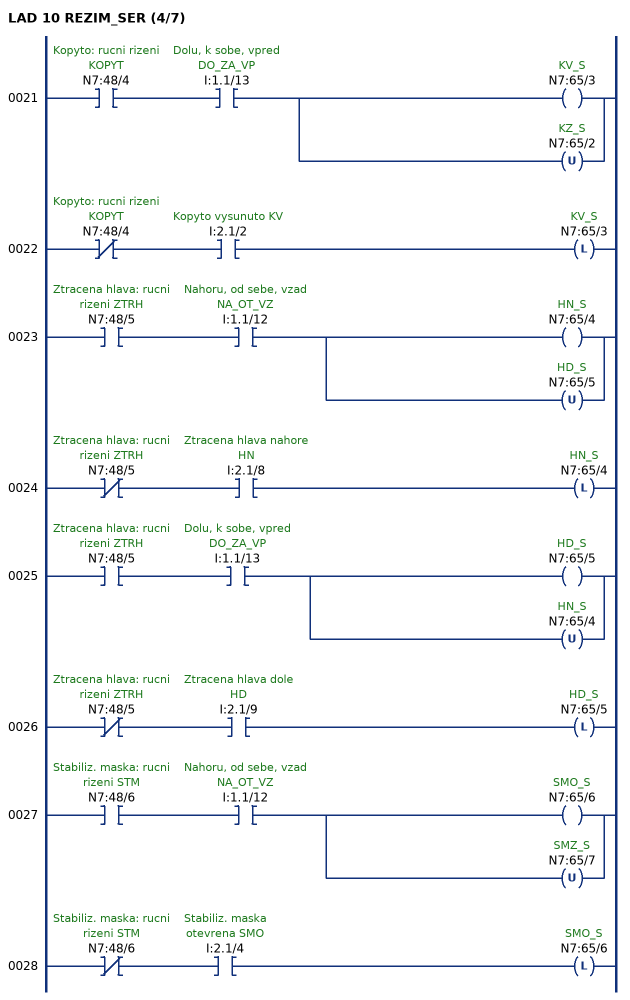
% Rung: 21 %
SOR XIC N7:48/4 XIC I:1.1/13 BST OTE N7:65/3 NXB OTU N7:65/2 BND EOR
%   N7:48/4  KOPYT  "Kopyto: rucni rizeni" %
%   I:1.1/13  DO_ZA_VP  "Dolu, k sobe, vpred" %
%   N7:65/3  KV_S %
%   N7:65/2  KZ_S %
% Rung: 22 %
SOR XIO N7:48/4 XIC I:2.1/2 OTL N7:65/3 EOR
%   N7:48/4  KOPYT  "Kopyto: rucni rizeni" %
%   I:2.1/2  KV  "Kopyto vysunuto" %
%   N7:65/3  KV_S %
% Rung: 23 %
SOR XIC N7:48/5 XIC I:1.1/12 BST OTE N7:65/4 NXB OTU N7:65/5 BND EOR
%   N7:48/5  ZTRH  "Ztracena hlava: rucni rizeni" %
%   I:1.1/12  NA_OT_VZ  "Nahoru, od sebe, vzad" %
%   N7:65/4  HN_S %
%   N7:65/5  HD_S %
% Rung: 24 %
SOR XIO N7:48/5 XIC I:2.1/8 OTL N7:65/4 EOR
%   N7:48/5  ZTRH  "Ztracena hlava: rucni rizeni" %
%   I:2.1/8  HN  "Ztracena hlava nahore" %
%   N7:65/4  HN_S %
% Rung: 25 %
SOR XIC N7:48/5 XIC I:1.1/13 BST OTE N7:65/5 NXB OTU N7:65/4 BND EOR
%   N7:48/5  ZTRH  "Ztracena hlava: rucni rizeni" %
%   I:1.1/13  DO_ZA_VP  "Dolu, k sobe, vpred" %
%   N7:65/5  HD_S %
%   N7:65/4  HN_S %
% Rung: 26 %
SOR XIO N7:48/5 XIC I:2.1/9 OTL N7:65/5 EOR
%   N7:48/5  ZTRH  "Ztracena hlava: rucni rizeni" %
%   I:2.1/9  HD  "Ztracena hlava dole" %
%   N7:65/5  HD_S %
% Rung: 27 %
SOR XIC N7:48/6 XIC I:1.1/12 BST OTE N7:65/6 NXB OTU N7:65/7 BND EOR
%   N7:48/6  STM  "Stabiliz. maska: rucni rizeni" %
%   I:1.1/12  NA_OT_VZ  "Nahoru, od sebe, vzad" %
%   N7:65/6  SMO_S %
%   N7:65/7  SMZ_S %
% Rung: 28 %
SOR XIO N7:48/6 XIC I:2.1/4 OTL N7:65/6 EOR
%   N7:48/6  STM  "Stabiliz. maska: rucni rizeni" %
%   I:2.1/4  SMO  "Stabiliz. maska otevrena" %
%   N7:65/6  SMO_S %

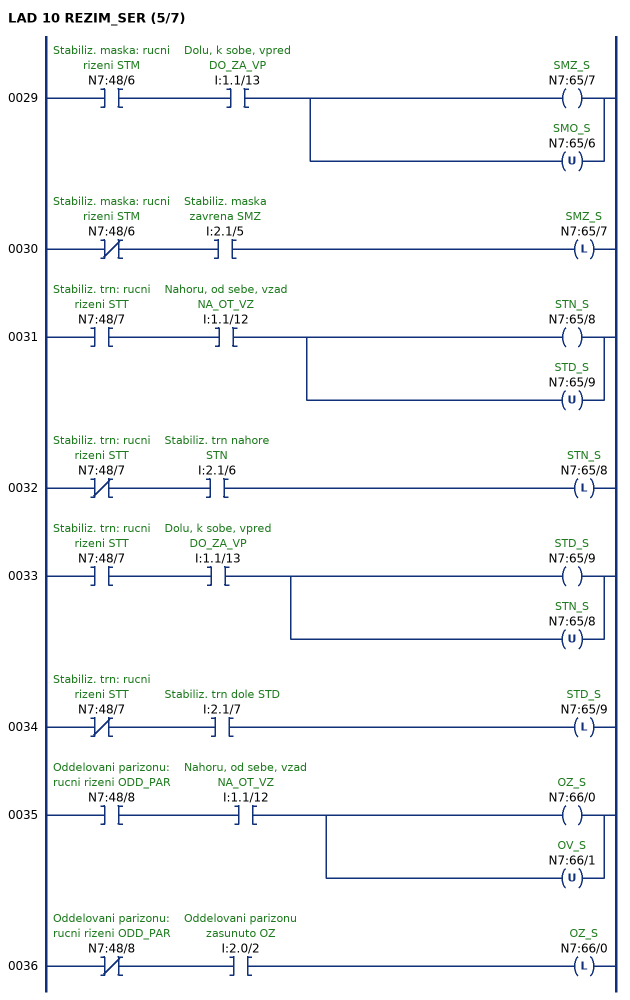
% Rung: 29 %
SOR XIC N7:48/6 XIC I:1.1/13 BST OTE N7:65/7 NXB OTU N7:65/6 BND EOR
%   N7:48/6  STM  "Stabiliz. maska: rucni rizeni" %
%   I:1.1/13  DO_ZA_VP  "Dolu, k sobe, vpred" %
%   N7:65/7  SMZ_S %
%   N7:65/6  SMO_S %
% Rung: 30 %
SOR XIO N7:48/6 XIC I:2.1/5 OTL N7:65/7 EOR
%   N7:48/6  STM  "Stabiliz. maska: rucni rizeni" %
%   I:2.1/5  SMZ  "Stabiliz. maska zavrena" %
%   N7:65/7  SMZ_S %
% Rung: 31 %
SOR XIC N7:48/7 XIC I:1.1/12 BST OTE N7:65/8 NXB OTU N7:65/9 BND EOR
%   N7:48/7  STT  "Stabiliz. trn: rucni rizeni" %
%   I:1.1/12  NA_OT_VZ  "Nahoru, od sebe, vzad" %
%   N7:65/8  STN_S %
%   N7:65/9  STD_S %
% Rung: 32 %
SOR XIO N7:48/7 XIC I:2.1/6 OTL N7:65/8 EOR
%   N7:48/7  STT  "Stabiliz. trn: rucni rizeni" %
%   I:2.1/6  STN  "Stabiliz. trn nahore" %
%   N7:65/8  STN_S %
% Rung: 33 %
SOR XIC N7:48/7 XIC I:1.1/13 BST OTE N7:65/9 NXB OTU N7:65/8 BND EOR
%   N7:48/7  STT  "Stabiliz. trn: rucni rizeni" %
%   I:1.1/13  DO_ZA_VP  "Dolu, k sobe, vpred" %
%   N7:65/9  STD_S %
%   N7:65/8  STN_S %
% Rung: 34 %
SOR XIO N7:48/7 XIC I:2.1/7 OTL N7:65/9 EOR
%   N7:48/7  STT  "Stabiliz. trn: rucni rizeni" %
%   I:2.1/7  STD  "Stabiliz. trn dole" %
%   N7:65/9  STD_S %
% Rung: 35 %
SOR XIC N7:48/8 XIC I:1.1/12 BST OTE N7:66/0 NXB OTU N7:66/1 BND EOR
%   N7:48/8  ODD_PAR  "Oddelovani parizonu: rucni rizeni" %
%   I:1.1/12  NA_OT_VZ  "Nahoru, od sebe, vzad" %
%   N7:66/0  OZ_S %
%   N7:66/1  OV_S %
% Rung: 36 %
SOR XIO N7:48/8 XIC I:2.0/2 OTL N7:66/0 EOR
%   N7:48/8  ODD_PAR  "Oddelovani parizonu: rucni rizeni" %
%   I:2.0/2  OZ  "Oddelovani parizonu zasunuto" %
%   N7:66/0  OZ_S %

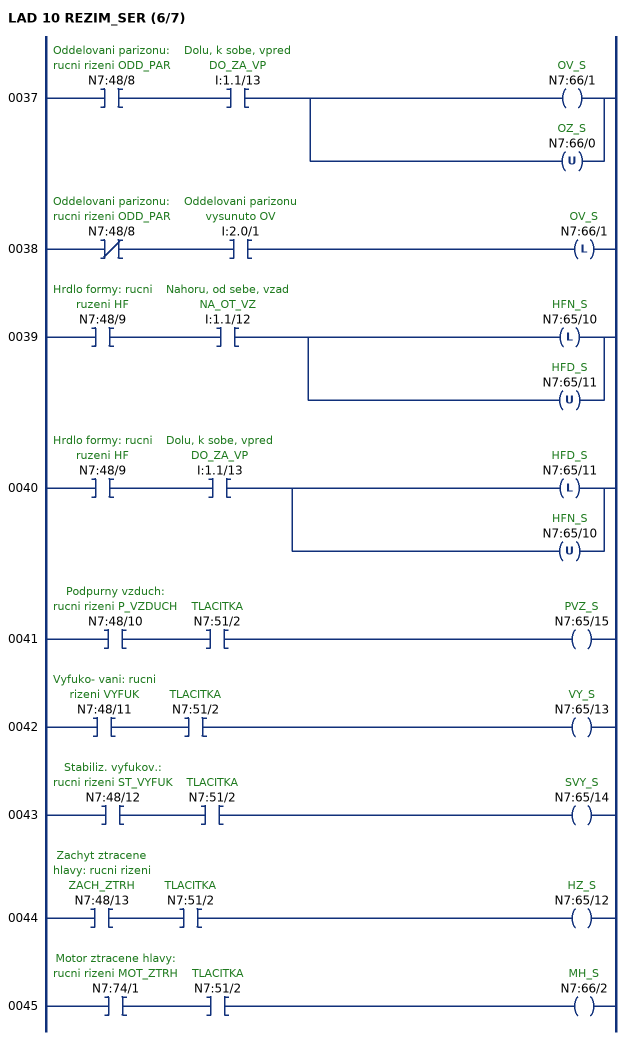
% Rung: 37 %
SOR XIC N7:48/8 XIC I:1.1/13 BST OTE N7:66/1 NXB OTU N7:66/0 BND EOR
%   N7:48/8  ODD_PAR  "Oddelovani parizonu: rucni rizeni" %
%   I:1.1/13  DO_ZA_VP  "Dolu, k sobe, vpred" %
%   N7:66/1  OV_S %
%   N7:66/0  OZ_S %
% Rung: 38 %
SOR XIO N7:48/8 XIC I:2.0/1 OTL N7:66/1 EOR
%   N7:48/8  ODD_PAR  "Oddelovani parizonu: rucni rizeni" %
%   I:2.0/1  OV  "Oddelovani parizonu vysunuto" %
%   N7:66/1  OV_S %
% Rung: 39 %
SOR XIC N7:48/9 XIC I:1.1/12 BST OTL N7:65/10 NXB OTU N7:65/11 BND EOR
%   N7:48/9  HF  "Hrdlo formy: rucni ruzeni" %
%   I:1.1/12  NA_OT_VZ  "Nahoru, od sebe, vzad" %
%   N7:65/10  HFN_S %
%   N7:65/11  HFD_S %
% Rung: 40 %
SOR XIC N7:48/9 XIC I:1.1/13 BST OTL N7:65/11 NXB OTU N7:65/10 BND EOR
%   N7:48/9  HF  "Hrdlo formy: rucni ruzeni" %
%   I:1.1/13  DO_ZA_VP  "Dolu, k sobe, vpred" %
%   N7:65/11  HFD_S %
%   N7:65/10  HFN_S %
% Rung: 41 %
SOR XIC N7:48/10 XIC N7:51/2 OTE N7:65/15 EOR
%   N7:48/10  P_VZDUCH  "Podpurny vzduch: rucni rizeni" %
%   N7:51/2  TLACITKA %
%   N7:65/15  PVZ_S %
% Rung: 42 %
SOR XIC N7:48/11 XIC N7:51/2 OTE N7:65/13 EOR
%   N7:48/11  VYFUK  "Vyfuko- vani: rucni rizeni" %
%   N7:51/2  TLACITKA %
%   N7:65/13  VY_S %
% Rung: 43 %
SOR XIC N7:48/12 XIC N7:51/2 OTE N7:65/14 EOR
%   N7:48/12  ST_VYFUK  "Stabiliz. vyfukov.: rucni rizeni" %
%   N7:51/2  TLACITKA %
%   N7:65/14  SVY_S %
% Rung: 44 %
SOR XIC N7:48/13 XIC N7:51/2 OTE N7:65/12 EOR
%   N7:48/13  ZACH_ZTRH  "Zachyt ztracene hlavy: rucni rizeni" %
%   N7:51/2  TLACITKA %
%   N7:65/12  HZ_S %
% Rung: 45 %
SOR XIC N7:74/1 XIC N7:51/2 OTE N7:66/2 EOR
%   N7:74/1  MOT_ZTRH  "Motor ztracene hlavy: rucni rizeni" %
%   N7:51/2  TLACITKA %
%   N7:66/2  MH_S %

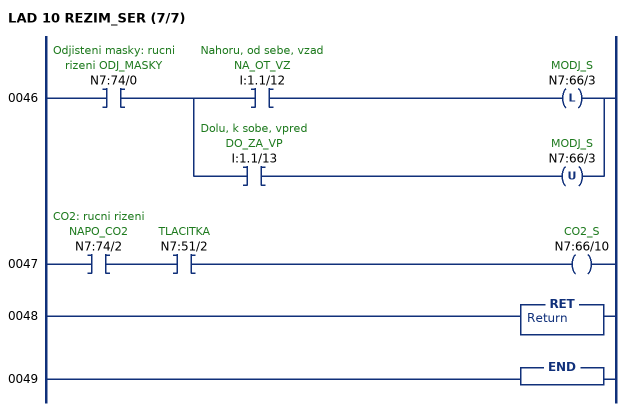
% Rung: 46 %
SOR XIC N7:74/0 BST XIC I:1.1/12 OTL N7:66/3 NXB XIC I:1.1/13 OTU N7:66/3 BND EOR
%   N7:74/0  ODJ_MASKY  "Odjisteni masky: rucni rizeni" %
%   I:1.1/12  NA_OT_VZ  "Nahoru, od sebe, vzad" %
%   N7:66/3  MODJ_S %
%   I:1.1/13  DO_ZA_VP  "Dolu, k sobe, vpred" %
% Rung: 47 %
SOR XIC N7:74/2 XIC N7:51/2 OTE N7:66/10 EOR
%   N7:74/2  NAPO_CO2  "CO2: rucni rizeni" %
%   N7:51/2  TLACITKA %
%   N7:66/10  CO2_S %
% Rung: 48 %
SOR RET EOR
% Rung: 49 %
SOR END EOR

LADDER 11 "REZIM_RUC"
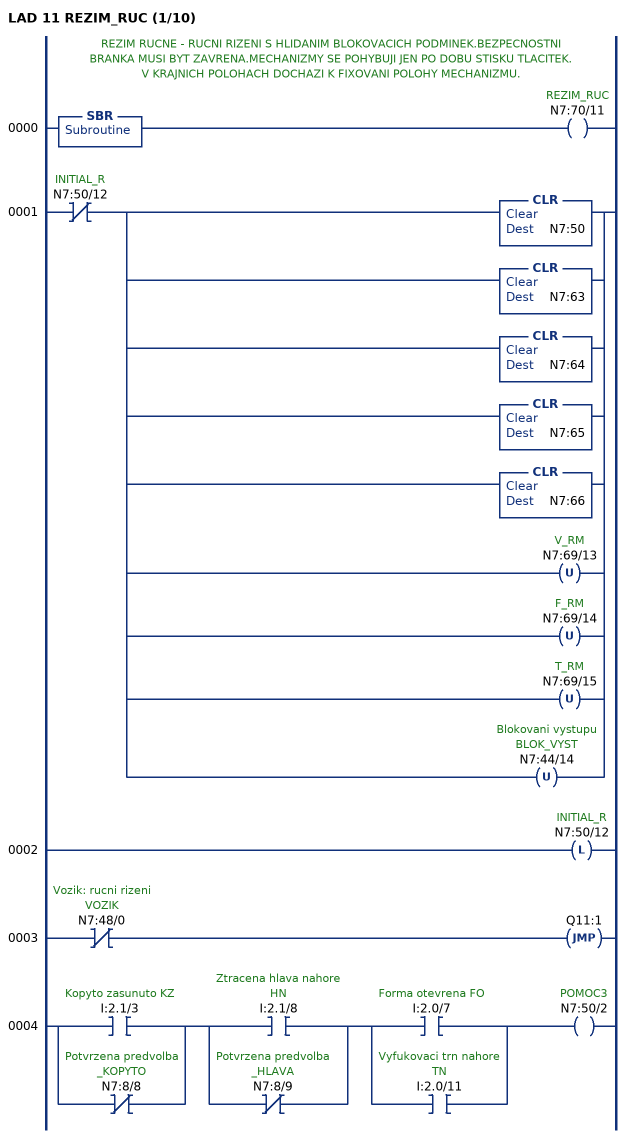
% Rung: 0 %
% REZIM RUCNE - RUCNI RIZENI S HLIDANIM BLOKOVACICH PODMINEK.BEZPECNOSTNI
% BRANKA MUSI BYT ZAVRENA.MECHANIZMY SE POHYBUJI JEN PO DOBU STISKU TLACITEK.
% V KRAJNICH POLOHACH DOCHAZI K FIXOVANI POLOHY MECHANIZMU. %
SOR SBR OTE N7:70/11 EOR
%   N7:70/11  REZIM_RUC %
% Rung: 1 %
SOR XIO N7:50/12 BST CLR N7:50 NXB CLR N7:63 NXB CLR N7:64 NXB CLR N7:65 NXB CLR N7:66 NXB OTU N7:69/13 NXB OTU N7:69/14 NXB OTU N7:69/15 NXB OTU N7:44/14 BND EOR
%   N7:50/12  INITIAL_R %
%   CLR N7:50  "Pomocne merkry" %
%   CLR N7:63  "Merkry vystupu rucniho rezimu" %
%   CLR N7:64  "Merkry vystupu rucniho rezimu" %
%   CLR N7:65  "Merkry vystupu rezimu serizovani" %
%   CLR N7:66  "Merkry vystupu rezimu serizovani" %
%   N7:69/13  V_RM %
%   N7:69/14  F_RM %
%   N7:69/15  T_RM %
%   N7:44/14  BLOK_VYST  "Blokovani vystupu" %
% Rung: 2 %
SOR OTL N7:50/12 EOR
%   N7:50/12  INITIAL_R %
% Rung: 3 %
SOR XIO N7:48/0 JMP Q11:1 EOR
%   N7:48/0  VOZIK  "Vozik: rucni rizeni" %
% Rung: 4 %
SOR BST XIC I:2.1/3 NXB XIO N7:8/8 BND BST XIC I:2.1/8 NXB XIO N7:8/9 BND BST XIC I:2.0/7 NXB XIC I:2.0/11 BND OTE N7:50/2 EOR
%   I:2.1/3  KZ  "Kopyto zasunuto" %
%   N7:8/8  _KOPYTO  "Potvrzena predvolba" %
%   I:2.1/8  HN  "Ztracena hlava nahore" %
%   N7:8/9  _HLAVA  "Potvrzena predvolba" %
%   I:2.0/7  FO  "Forma otevrena" %
%   I:2.0/11  TN  "Vyfukovaci trn nahore" %
%   N7:50/2  POMOC3 %

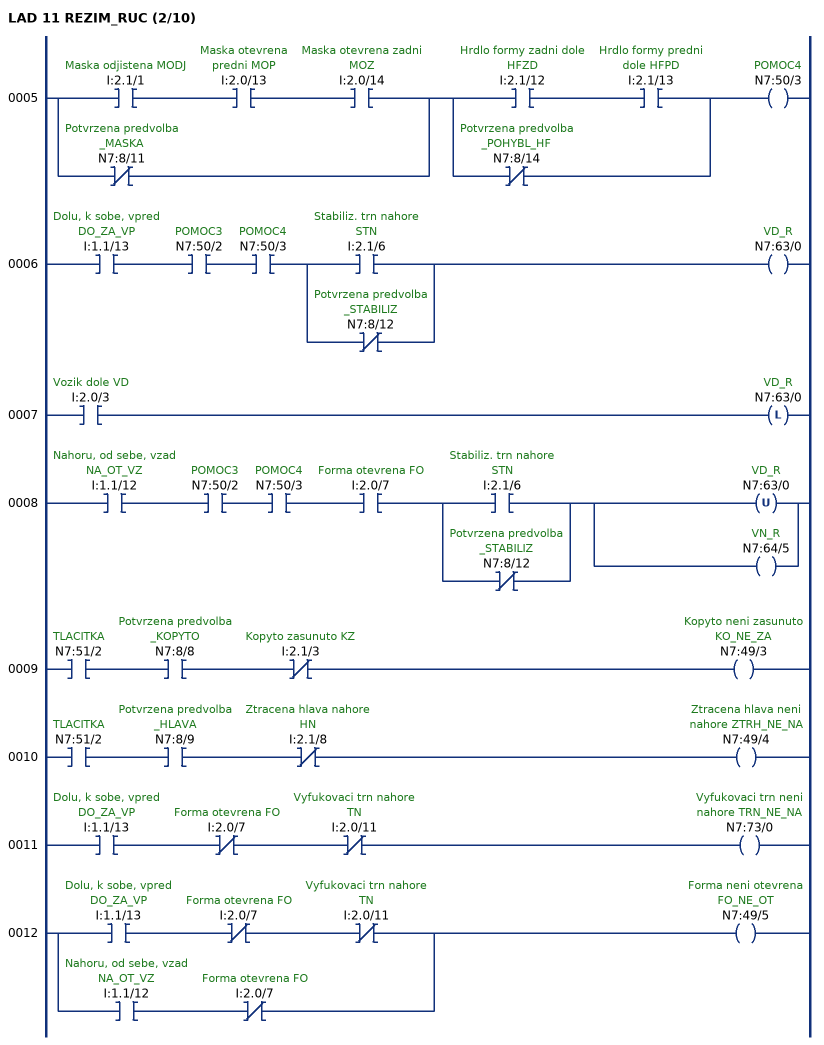
% Rung: 5 %
SOR BST XIC I:2.1/1 XIC I:2.0/13 XIC I:2.0/14 NXB XIO N7:8/11 BND BST XIC I:2.1/12 XIC I:2.1/13 NXB XIO N7:8/14 BND OTE N7:50/3 EOR
%   I:2.1/1  MODJ  "Maska odjistena" %
%   I:2.0/13  MOP  "Maska otevrena predni" %
%   I:2.0/14  MOZ  "Maska otevrena zadni" %
%   N7:8/11  _MASKA  "Potvrzena predvolba" %
%   I:2.1/12  HFZD  "Hrdlo formy zadni dole" %
%   I:2.1/13  HFPD  "Hrdlo formy predni dole" %
%   N7:8/14  _POHYBL_HF  "Potvrzena predvolba" %
%   N7:50/3  POMOC4 %
% Rung: 6 %
SOR XIC I:1.1/13 XIC N7:50/2 XIC N7:50/3 BST XIC I:2.1/6 NXB XIO N7:8/12 BND OTE N7:63/0 EOR
%   I:1.1/13  DO_ZA_VP  "Dolu, k sobe, vpred" %
%   N7:50/2  POMOC3 %
%   N7:50/3  POMOC4 %
%   I:2.1/6  STN  "Stabiliz. trn nahore" %
%   N7:8/12  _STABILIZ  "Potvrzena predvolba" %
%   N7:63/0  VD_R %
% Rung: 7 %
SOR XIC I:2.0/3 OTL N7:63/0 EOR
%   I:2.0/3  VD  "Vozik dole" %
%   N7:63/0  VD_R %
% Rung: 8 %
SOR XIC I:1.1/12 XIC N7:50/2 XIC N7:50/3 XIC I:2.0/7 BST XIC I:2.1/6 NXB XIO N7:8/12 BND BST OTU N7:63/0 NXB OTE N7:64/5 BND EOR
%   I:1.1/12  NA_OT_VZ  "Nahoru, od sebe, vzad" %
%   N7:50/2  POMOC3 %
%   N7:50/3  POMOC4 %
%   I:2.0/7  FO  "Forma otevrena" %
%   I:2.1/6  STN  "Stabiliz. trn nahore" %
%   N7:8/12  _STABILIZ  "Potvrzena predvolba" %
%   N7:63/0  VD_R %
%   N7:64/5  VN_R %
% Rung: 9 %
SOR XIC N7:51/2 XIC N7:8/8 XIO I:2.1/3 OTE N7:49/3 EOR
%   N7:51/2  TLACITKA %
%   N7:8/8  _KOPYTO  "Potvrzena predvolba" %
%   I:2.1/3  KZ  "Kopyto zasunuto" %
%   N7:49/3  KO_NE_ZA  "Kopyto neni zasunuto" %
% Rung: 10 %
SOR XIC N7:51/2 XIC N7:8/9 XIO I:2.1/8 OTE N7:49/4 EOR
%   N7:51/2  TLACITKA %
%   N7:8/9  _HLAVA  "Potvrzena predvolba" %
%   I:2.1/8  HN  "Ztracena hlava nahore" %
%   N7:49/4  ZTRH_NE_NA  "Ztracena hlava neni nahore" %
% Rung: 11 %
SOR XIC I:1.1/13 XIO I:2.0/7 XIO I:2.0/11 OTE N7:73/0 EOR
%   I:1.1/13  DO_ZA_VP  "Dolu, k sobe, vpred" %
%   I:2.0/7  FO  "Forma otevrena" %
%   I:2.0/11  TN  "Vyfukovaci trn nahore" %
%   N7:73/0  TRN_NE_NA  "Vyfukovaci trn neni nahore" %
% Rung: 12 %
SOR BST XIC I:1.1/13 XIO I:2.0/7 XIO I:2.0/11 NXB XIC I:1.1/12 XIO I:2.0/7 BND OTE N7:49/5 EOR
%   I:1.1/13  DO_ZA_VP  "Dolu, k sobe, vpred" %
%   I:2.0/7  FO  "Forma otevrena" %
%   I:2.0/11  TN  "Vyfukovaci trn nahore" %
%   I:1.1/12  NA_OT_VZ  "Nahoru, od sebe, vzad" %
%   N7:49/5  FO_NE_OT  "Forma neni otevrena" %

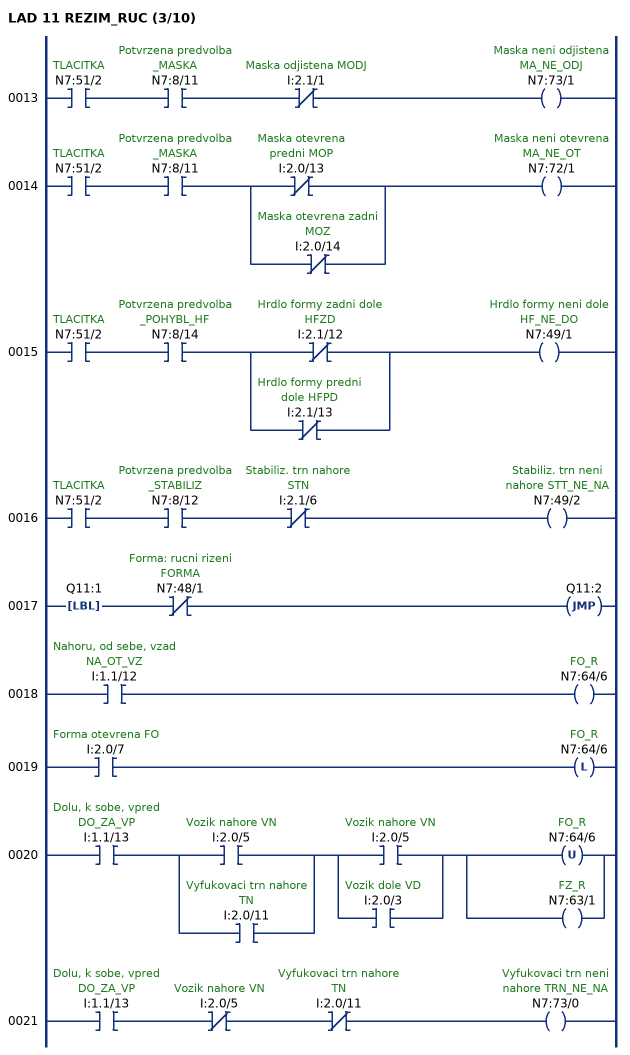
% Rung: 13 %
SOR XIC N7:51/2 XIC N7:8/11 XIO I:2.1/1 OTE N7:73/1 EOR
%   N7:51/2  TLACITKA %
%   N7:8/11  _MASKA  "Potvrzena predvolba" %
%   I:2.1/1  MODJ  "Maska odjistena" %
%   N7:73/1  MA_NE_ODJ  "Maska neni odjistena" %
% Rung: 14 %
SOR XIC N7:51/2 XIC N7:8/11 BST XIO I:2.0/13 NXB XIO I:2.0/14 BND OTE N7:72/1 EOR
%   N7:51/2  TLACITKA %
%   N7:8/11  _MASKA  "Potvrzena predvolba" %
%   I:2.0/13  MOP  "Maska otevrena predni" %
%   I:2.0/14  MOZ  "Maska otevrena zadni" %
%   N7:72/1  MA_NE_OT  "Maska neni otevrena" %
% Rung: 15 %
SOR XIC N7:51/2 XIC N7:8/14 BST XIO I:2.1/12 NXB XIO I:2.1/13 BND OTE N7:49/1 EOR
%   N7:51/2  TLACITKA %
%   N7:8/14  _POHYBL_HF  "Potvrzena predvolba" %
%   I:2.1/12  HFZD  "Hrdlo formy zadni dole" %
%   I:2.1/13  HFPD  "Hrdlo formy predni dole" %
%   N7:49/1  HF_NE_DO  "Hrdlo formy neni dole" %
% Rung: 16 %
SOR XIC N7:51/2 XIC N7:8/12 XIO I:2.1/6 OTE N7:49/2 EOR
%   N7:51/2  TLACITKA %
%   N7:8/12  _STABILIZ  "Potvrzena predvolba" %
%   I:2.1/6  STN  "Stabiliz. trn nahore" %
%   N7:49/2  STT_NE_NA  "Stabiliz. trn neni nahore" %
% Rung: 17 %
SOR LBL Q11:1 XIO N7:48/1 JMP Q11:2 EOR
%   N7:48/1  FORMA  "Forma: rucni rizeni" %
% Rung: 18 %
SOR XIC I:1.1/12 OTE N7:64/6 EOR
%   I:1.1/12  NA_OT_VZ  "Nahoru, od sebe, vzad" %
%   N7:64/6  FO_R %
% Rung: 19 %
SOR XIC I:2.0/7 OTL N7:64/6 EOR
%   I:2.0/7  FO  "Forma otevrena" %
%   N7:64/6  FO_R %
% Rung: 20 %
SOR XIC I:1.1/13 BST XIC I:2.0/5 NXB XIC I:2.0/11 BND BST XIC I:2.0/5 NXB XIC I:2.0/3 BND BST OTU N7:64/6 NXB OTE N7:63/1 BND EOR
%   I:1.1/13  DO_ZA_VP  "Dolu, k sobe, vpred" %
%   I:2.0/5  VN  "Vozik nahore" %
%   I:2.0/11  TN  "Vyfukovaci trn nahore" %
%   I:2.0/3  VD  "Vozik dole" %
%   N7:64/6  FO_R %
%   N7:63/1  FZ_R %
% Rung: 21 %
SOR XIC I:1.1/13 XIO I:2.0/5 XIO I:2.0/11 OTE N7:73/0 EOR
%   I:1.1/13  DO_ZA_VP  "Dolu, k sobe, vpred" %
%   I:2.0/5  VN  "Vozik nahore" %
%   I:2.0/11  TN  "Vyfukovaci trn nahore" %
%   N7:73/0  TRN_NE_NA  "Vyfukovaci trn neni nahore" %

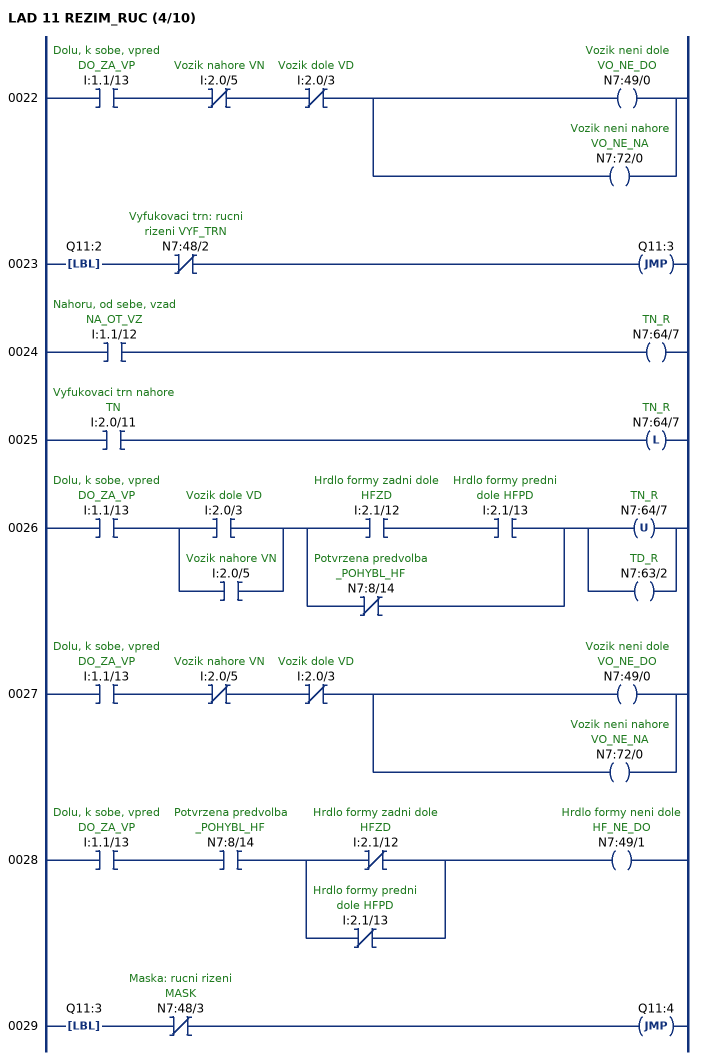
% Rung: 22 %
SOR XIC I:1.1/13 XIO I:2.0/5 XIO I:2.0/3 BST OTE N7:49/0 NXB OTE N7:72/0 BND EOR
%   I:1.1/13  DO_ZA_VP  "Dolu, k sobe, vpred" %
%   I:2.0/5  VN  "Vozik nahore" %
%   I:2.0/3  VD  "Vozik dole" %
%   N7:49/0  VO_NE_DO  "Vozik neni dole" %
%   N7:72/0  VO_NE_NA  "Vozik neni nahore" %
% Rung: 23 %
SOR LBL Q11:2 XIO N7:48/2 JMP Q11:3 EOR
%   N7:48/2  VYF_TRN  "Vyfukovaci trn: rucni rizeni" %
% Rung: 24 %
SOR XIC I:1.1/12 OTE N7:64/7 EOR
%   I:1.1/12  NA_OT_VZ  "Nahoru, od sebe, vzad" %
%   N7:64/7  TN_R %
% Rung: 25 %
SOR XIC I:2.0/11 OTL N7:64/7 EOR
%   I:2.0/11  TN  "Vyfukovaci trn nahore" %
%   N7:64/7  TN_R %
% Rung: 26 %
SOR XIC I:1.1/13 BST XIC I:2.0/3 NXB XIC I:2.0/5 BND BST XIC I:2.1/12 XIC I:2.1/13 NXB XIO N7:8/14 BND BST OTU N7:64/7 NXB OTE N7:63/2 BND EOR
%   I:1.1/13  DO_ZA_VP  "Dolu, k sobe, vpred" %
%   I:2.0/3  VD  "Vozik dole" %
%   I:2.0/5  VN  "Vozik nahore" %
%   I:2.1/12  HFZD  "Hrdlo formy zadni dole" %
%   I:2.1/13  HFPD  "Hrdlo formy predni dole" %
%   N7:8/14  _POHYBL_HF  "Potvrzena predvolba" %
%   N7:64/7  TN_R %
%   N7:63/2  TD_R %
% Rung: 27 %
SOR XIC I:1.1/13 XIO I:2.0/5 XIO I:2.0/3 BST OTE N7:49/0 NXB OTE N7:72/0 BND EOR
%   I:1.1/13  DO_ZA_VP  "Dolu, k sobe, vpred" %
%   I:2.0/5  VN  "Vozik nahore" %
%   I:2.0/3  VD  "Vozik dole" %
%   N7:49/0  VO_NE_DO  "Vozik neni dole" %
%   N7:72/0  VO_NE_NA  "Vozik neni nahore" %
% Rung: 28 %
SOR XIC I:1.1/13 XIC N7:8/14 BST XIO I:2.1/12 NXB XIO I:2.1/13 BND OTE N7:49/1 EOR
%   I:1.1/13  DO_ZA_VP  "Dolu, k sobe, vpred" %
%   N7:8/14  _POHYBL_HF  "Potvrzena predvolba" %
%   I:2.1/12  HFZD  "Hrdlo formy zadni dole" %
%   I:2.1/13  HFPD  "Hrdlo formy predni dole" %
%   N7:49/1  HF_NE_DO  "Hrdlo formy neni dole" %
% Rung: 29 %
SOR LBL Q11:3 XIO N7:48/3 JMP Q11:4 EOR
%   N7:48/3  MASK  "Maska: rucni rizeni" %

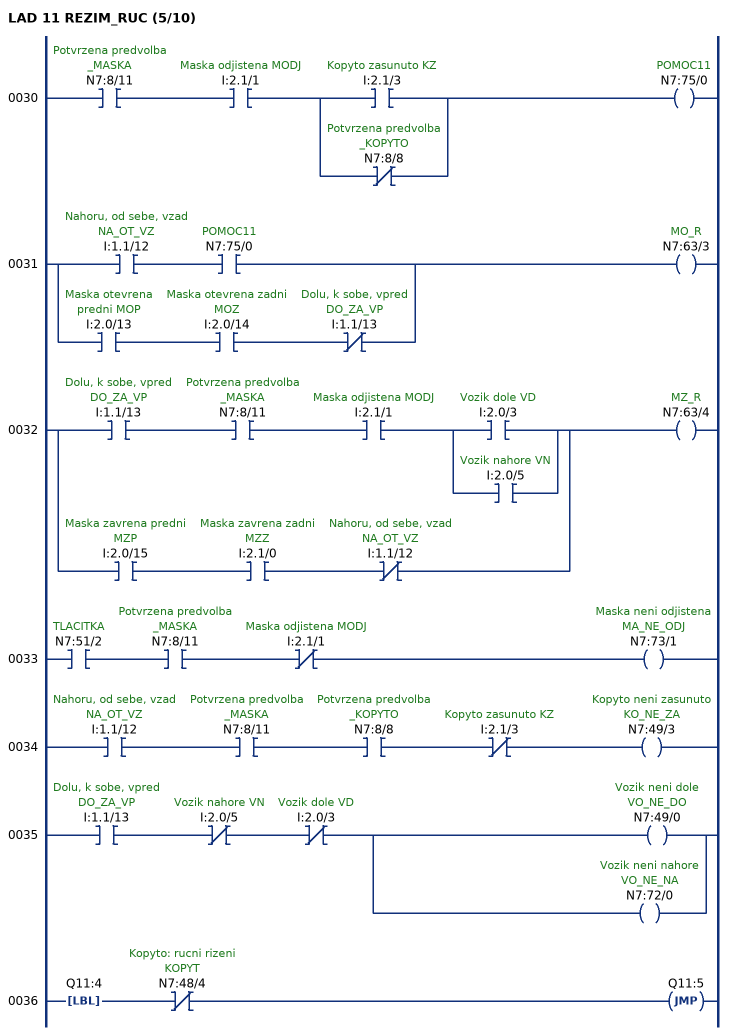
% Rung: 30 %
SOR XIC N7:8/11 XIC I:2.1/1 BST XIC I:2.1/3 NXB XIO N7:8/8 BND OTE N7:75/0 EOR
%   N7:8/11  _MASKA  "Potvrzena predvolba" %
%   I:2.1/1  MODJ  "Maska odjistena" %
%   I:2.1/3  KZ  "Kopyto zasunuto" %
%   N7:8/8  _KOPYTO  "Potvrzena predvolba" %
%   N7:75/0  POMOC11 %
% Rung: 31 %
SOR BST XIC I:1.1/12 XIC N7:75/0 NXB XIC I:2.0/13 XIC I:2.0/14 XIO I:1.1/13 BND OTE N7:63/3 EOR
%   I:1.1/12  NA_OT_VZ  "Nahoru, od sebe, vzad" %
%   N7:75/0  POMOC11 %
%   I:2.0/13  MOP  "Maska otevrena predni" %
%   I:2.0/14  MOZ  "Maska otevrena zadni" %
%   I:1.1/13  DO_ZA_VP  "Dolu, k sobe, vpred" %
%   N7:63/3  MO_R %
% Rung: 32 %
SOR BST XIC I:1.1/13 XIC N7:8/11 XIC I:2.1/1 BST XIC I:2.0/3 NXB XIC I:2.0/5 BND NXB XIC I:2.0/15 XIC I:2.1/0 XIO I:1.1/12 BND OTE N7:63/4 EOR
%   I:1.1/13  DO_ZA_VP  "Dolu, k sobe, vpred" %
%   N7:8/11  _MASKA  "Potvrzena predvolba" %
%   I:2.1/1  MODJ  "Maska odjistena" %
%   I:2.0/3  VD  "Vozik dole" %
%   I:2.0/5  VN  "Vozik nahore" %
%   I:2.0/15  MZP  "Maska zavrena predni" %
%   I:2.1/0  MZZ  "Maska zavrena zadni" %
%   I:1.1/12  NA_OT_VZ  "Nahoru, od sebe, vzad" %
%   N7:63/4  MZ_R %
% Rung: 33 %
SOR XIC N7:51/2 XIC N7:8/11 XIO I:2.1/1 OTE N7:73/1 EOR
%   N7:51/2  TLACITKA %
%   N7:8/11  _MASKA  "Potvrzena predvolba" %
%   I:2.1/1  MODJ  "Maska odjistena" %
%   N7:73/1  MA_NE_ODJ  "Maska neni odjistena" %
% Rung: 34 %
SOR XIC I:1.1/12 XIC N7:8/11 XIC N7:8/8 XIO I:2.1/3 OTE N7:49/3 EOR
%   I:1.1/12  NA_OT_VZ  "Nahoru, od sebe, vzad" %
%   N7:8/11  _MASKA  "Potvrzena predvolba" %
%   N7:8/8  _KOPYTO  "Potvrzena predvolba" %
%   I:2.1/3  KZ  "Kopyto zasunuto" %
%   N7:49/3  KO_NE_ZA  "Kopyto neni zasunuto" %
% Rung: 35 %
SOR XIC I:1.1/13 XIO I:2.0/5 XIO I:2.0/3 BST OTE N7:49/0 NXB OTE N7:72/0 BND EOR
%   I:1.1/13  DO_ZA_VP  "Dolu, k sobe, vpred" %
%   I:2.0/5  VN  "Vozik nahore" %
%   I:2.0/3  VD  "Vozik dole" %
%   N7:49/0  VO_NE_DO  "Vozik neni dole" %
%   N7:72/0  VO_NE_NA  "Vozik neni nahore" %
% Rung: 36 %
SOR LBL Q11:4 XIO N7:48/4 JMP Q11:5 EOR
%   N7:48/4  KOPYT  "Kopyto: rucni rizeni" %

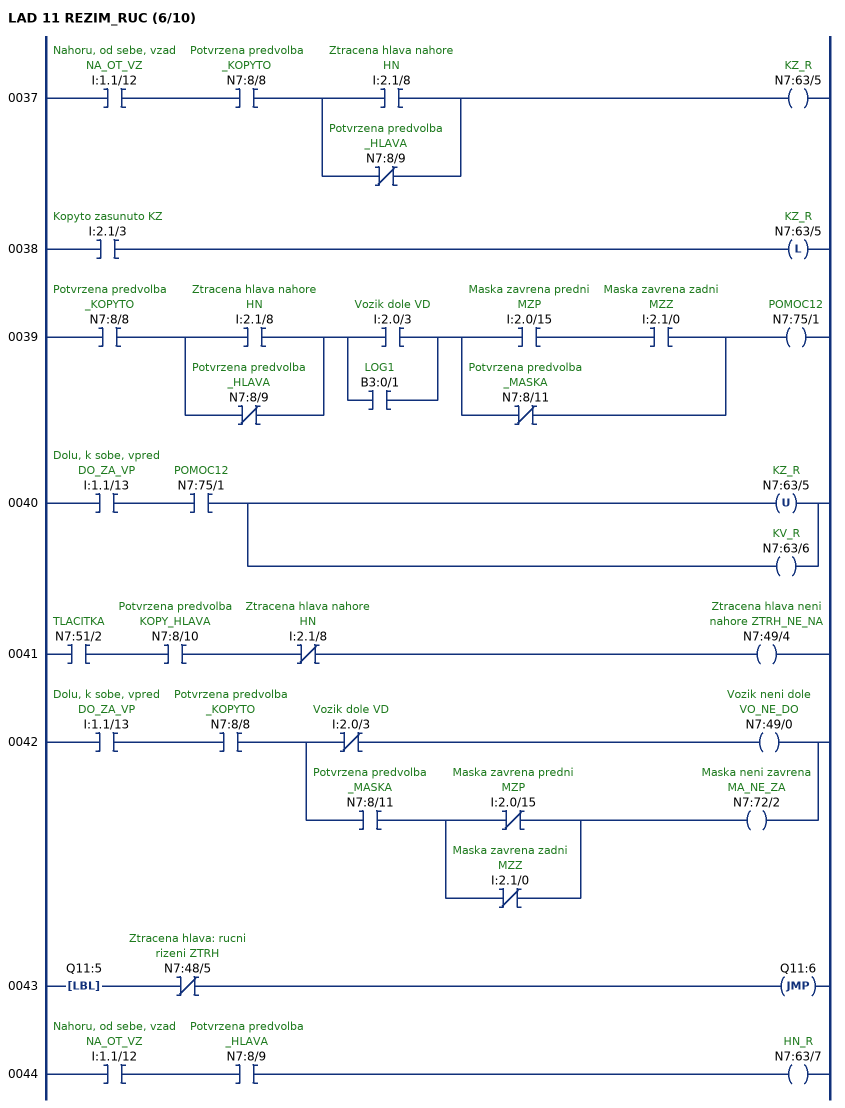
% Rung: 37 %
SOR XIC I:1.1/12 XIC N7:8/8 BST XIC I:2.1/8 NXB XIO N7:8/9 BND OTE N7:63/5 EOR
%   I:1.1/12  NA_OT_VZ  "Nahoru, od sebe, vzad" %
%   N7:8/8  _KOPYTO  "Potvrzena predvolba" %
%   I:2.1/8  HN  "Ztracena hlava nahore" %
%   N7:8/9  _HLAVA  "Potvrzena predvolba" %
%   N7:63/5  KZ_R %
% Rung: 38 %
SOR XIC I:2.1/3 OTL N7:63/5 EOR
%   I:2.1/3  KZ  "Kopyto zasunuto" %
%   N7:63/5  KZ_R %
% Rung: 39 %
SOR XIC N7:8/8 BST XIC I:2.1/8 NXB XIO N7:8/9 BND BST XIC I:2.0/3 NXB XIC B3:0/1 BND BST XIC I:2.0/15 XIC I:2.1/0 NXB XIO N7:8/11 BND OTE N7:75/1 EOR
%   N7:8/8  _KOPYTO  "Potvrzena predvolba" %
%   I:2.1/8  HN  "Ztracena hlava nahore" %
%   N7:8/9  _HLAVA  "Potvrzena predvolba" %
%   I:2.0/3  VD  "Vozik dole" %
%   B3:0/1  LOG1 %
%   I:2.0/15  MZP  "Maska zavrena predni" %
%   I:2.1/0  MZZ  "Maska zavrena zadni" %
%   N7:8/11  _MASKA  "Potvrzena predvolba" %
%   N7:75/1  POMOC12 %
% Rung: 40 %
SOR XIC I:1.1/13 XIC N7:75/1 BST OTU N7:63/5 NXB OTE N7:63/6 BND EOR
%   I:1.1/13  DO_ZA_VP  "Dolu, k sobe, vpred" %
%   N7:75/1  POMOC12 %
%   N7:63/5  KZ_R %
%   N7:63/6  KV_R %
% Rung: 41 %
SOR XIC N7:51/2 XIC N7:8/10 XIO I:2.1/8 OTE N7:49/4 EOR
%   N7:51/2  TLACITKA %
%   N7:8/10  KOPY_HLAVA  "Potvrzena predvolba" %
%   I:2.1/8  HN  "Ztracena hlava nahore" %
%   N7:49/4  ZTRH_NE_NA  "Ztracena hlava neni nahore" %
% Rung: 42 %
SOR XIC I:1.1/13 XIC N7:8/8 BST XIO I:2.0/3 OTE N7:49/0 NXB XIC N7:8/11 BST XIO I:2.0/15 NXB XIO I:2.1/0 BND OTE N7:72/2 BND EOR
%   I:1.1/13  DO_ZA_VP  "Dolu, k sobe, vpred" %
%   N7:8/8  _KOPYTO  "Potvrzena predvolba" %
%   I:2.0/3  VD  "Vozik dole" %
%   N7:49/0  VO_NE_DO  "Vozik neni dole" %
%   N7:8/11  _MASKA  "Potvrzena predvolba" %
%   I:2.0/15  MZP  "Maska zavrena predni" %
%   I:2.1/0  MZZ  "Maska zavrena zadni" %
%   N7:72/2  MA_NE_ZA  "Maska neni zavrena" %
% Rung: 43 %
SOR LBL Q11:5 XIO N7:48/5 JMP Q11:6 EOR
%   N7:48/5  ZTRH  "Ztracena hlava: rucni rizeni" %
% Rung: 44 %
SOR XIC I:1.1/12 XIC N7:8/9 OTE N7:63/7 EOR
%   I:1.1/12  NA_OT_VZ  "Nahoru, od sebe, vzad" %
%   N7:8/9  _HLAVA  "Potvrzena predvolba" %
%   N7:63/7  HN_R %

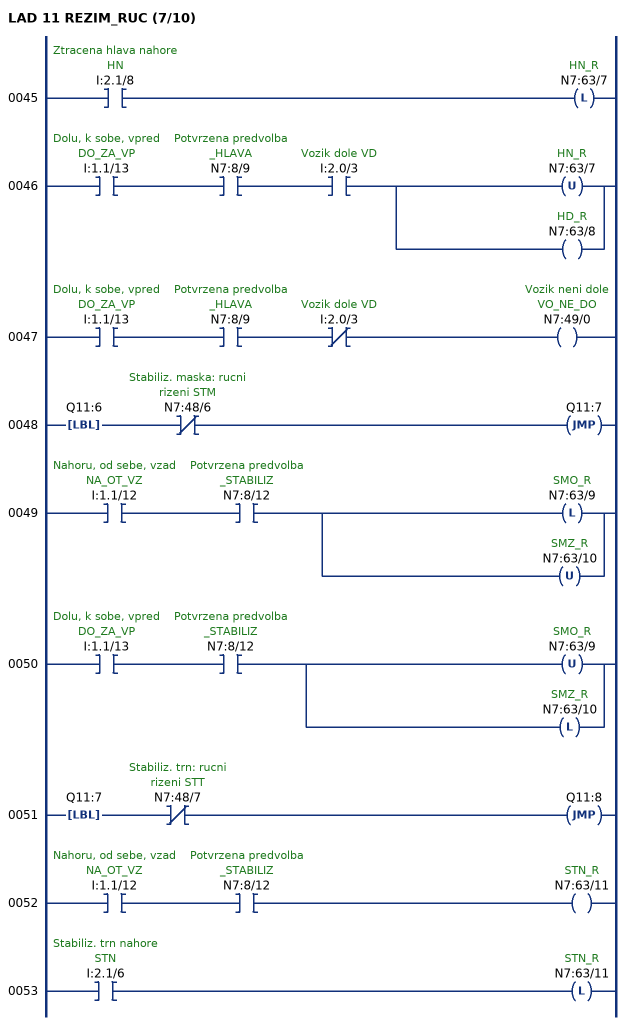
% Rung: 45 %
SOR XIC I:2.1/8 OTL N7:63/7 EOR
%   I:2.1/8  HN  "Ztracena hlava nahore" %
%   N7:63/7  HN_R %
% Rung: 46 %
SOR XIC I:1.1/13 XIC N7:8/9 XIC I:2.0/3 BST OTU N7:63/7 NXB OTE N7:63/8 BND EOR
%   I:1.1/13  DO_ZA_VP  "Dolu, k sobe, vpred" %
%   N7:8/9  _HLAVA  "Potvrzena predvolba" %
%   I:2.0/3  VD  "Vozik dole" %
%   N7:63/7  HN_R %
%   N7:63/8  HD_R %
% Rung: 47 %
SOR XIC I:1.1/13 XIC N7:8/9 XIO I:2.0/3 OTE N7:49/0 EOR
%   I:1.1/13  DO_ZA_VP  "Dolu, k sobe, vpred" %
%   N7:8/9  _HLAVA  "Potvrzena predvolba" %
%   I:2.0/3  VD  "Vozik dole" %
%   N7:49/0  VO_NE_DO  "Vozik neni dole" %
% Rung: 48 %
SOR LBL Q11:6 XIO N7:48/6 JMP Q11:7 EOR
%   N7:48/6  STM  "Stabiliz. maska: rucni rizeni" %
% Rung: 49 %
SOR XIC I:1.1/12 XIC N7:8/12 BST OTL N7:63/9 NXB OTU N7:63/10 BND EOR
%   I:1.1/12  NA_OT_VZ  "Nahoru, od sebe, vzad" %
%   N7:8/12  _STABILIZ  "Potvrzena predvolba" %
%   N7:63/9  SMO_R %
%   N7:63/10  SMZ_R %
% Rung: 50 %
SOR XIC I:1.1/13 XIC N7:8/12 BST OTU N7:63/9 NXB OTL N7:63/10 BND EOR
%   I:1.1/13  DO_ZA_VP  "Dolu, k sobe, vpred" %
%   N7:8/12  _STABILIZ  "Potvrzena predvolba" %
%   N7:63/9  SMO_R %
%   N7:63/10  SMZ_R %
% Rung: 51 %
SOR LBL Q11:7 XIO N7:48/7 JMP Q11:8 EOR
%   N7:48/7  STT  "Stabiliz. trn: rucni rizeni" %
% Rung: 52 %
SOR XIC I:1.1/12 XIC N7:8/12 OTE N7:63/11 EOR
%   I:1.1/12  NA_OT_VZ  "Nahoru, od sebe, vzad" %
%   N7:8/12  _STABILIZ  "Potvrzena predvolba" %
%   N7:63/11  STN_R %
% Rung: 53 %
SOR XIC I:2.1/6 OTL N7:63/11 EOR
%   I:2.1/6  STN  "Stabiliz. trn nahore" %
%   N7:63/11  STN_R %

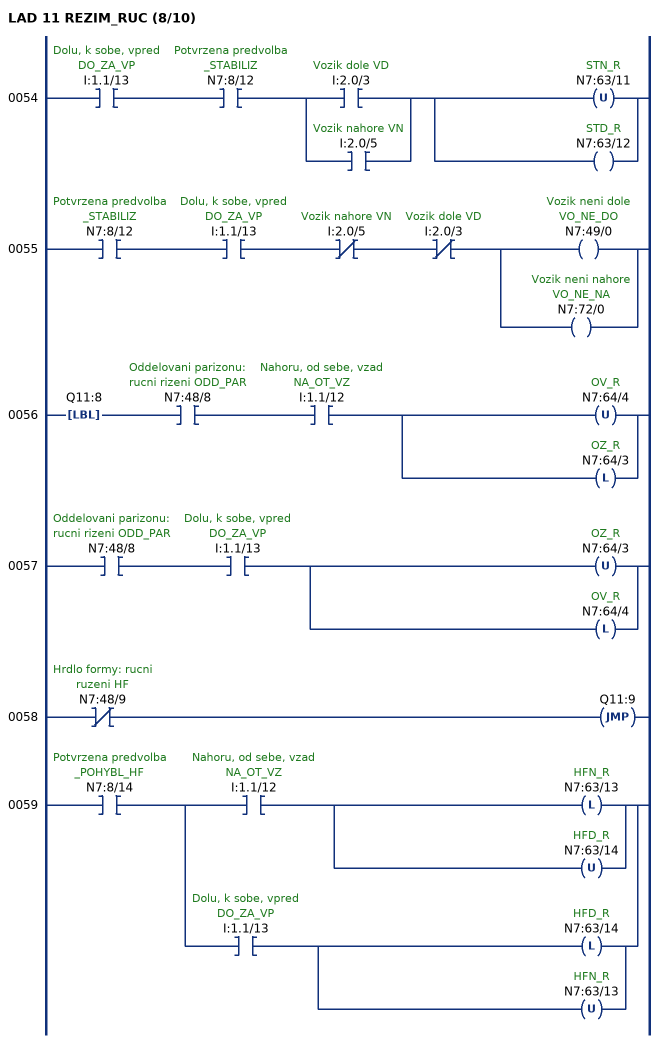
% Rung: 54 %
SOR XIC I:1.1/13 XIC N7:8/12 BST XIC I:2.0/3 NXB XIC I:2.0/5 BND BST OTU N7:63/11 NXB OTE N7:63/12 BND EOR
%   I:1.1/13  DO_ZA_VP  "Dolu, k sobe, vpred" %
%   N7:8/12  _STABILIZ  "Potvrzena predvolba" %
%   I:2.0/3  VD  "Vozik dole" %
%   I:2.0/5  VN  "Vozik nahore" %
%   N7:63/11  STN_R %
%   N7:63/12  STD_R %
% Rung: 55 %
SOR XIC N7:8/12 XIC I:1.1/13 XIO I:2.0/5 XIO I:2.0/3 BST OTE N7:49/0 NXB OTE N7:72/0 BND EOR
%   N7:8/12  _STABILIZ  "Potvrzena predvolba" %
%   I:1.1/13  DO_ZA_VP  "Dolu, k sobe, vpred" %
%   I:2.0/5  VN  "Vozik nahore" %
%   I:2.0/3  VD  "Vozik dole" %
%   N7:49/0  VO_NE_DO  "Vozik neni dole" %
%   N7:72/0  VO_NE_NA  "Vozik neni nahore" %
% Rung: 56 %
SOR LBL Q11:8 XIC N7:48/8 XIC I:1.1/12 BST OTU N7:64/4 NXB OTL N7:64/3 BND EOR
%   N7:48/8  ODD_PAR  "Oddelovani parizonu: rucni rizeni" %
%   I:1.1/12  NA_OT_VZ  "Nahoru, od sebe, vzad" %
%   N7:64/4  OV_R %
%   N7:64/3  OZ_R %
% Rung: 57 %
SOR XIC N7:48/8 XIC I:1.1/13 BST OTU N7:64/3 NXB OTL N7:64/4 BND EOR
%   N7:48/8  ODD_PAR  "Oddelovani parizonu: rucni rizeni" %
%   I:1.1/13  DO_ZA_VP  "Dolu, k sobe, vpred" %
%   N7:64/3  OZ_R %
%   N7:64/4  OV_R %
% Rung: 58 %
SOR XIO N7:48/9 JMP Q11:9 EOR
%   N7:48/9  HF  "Hrdlo formy: rucni ruzeni" %
% Rung: 59 %
SOR XIC N7:8/14 BST XIC I:1.1/12 BST OTL N7:63/13 NXB OTU N7:63/14 BND NXB XIC I:1.1/13 BST OTL N7:63/14 NXB OTU N7:63/13 BND BND EOR
%   N7:8/14  _POHYBL_HF  "Potvrzena predvolba" %
%   I:1.1/12  NA_OT_VZ  "Nahoru, od sebe, vzad" %
%   N7:63/13  HFN_R %
%   N7:63/14  HFD_R %
%   I:1.1/13  DO_ZA_VP  "Dolu, k sobe, vpred" %

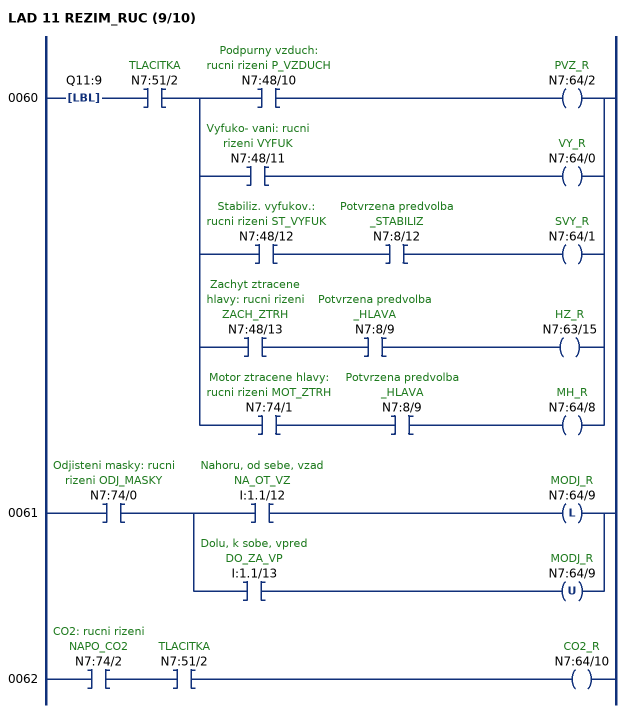
% Rung: 60 %
SOR LBL Q11:9 XIC N7:51/2 BST XIC N7:48/10 OTE N7:64/2 NXB BST XIC N7:48/11 OTE N7:64/0 NXB XIC N7:48/12 XIC N7:8/12 OTE N7:64/1 NXB XIC N7:48/13 XIC N7:8/9 OTE N7:63/15 NXB XIC N7:74/1 XIC N7:8/9 OTE N7:64/8 BND BND EOR
%   N7:51/2  TLACITKA %
%   N7:48/10  P_VZDUCH  "Podpurny vzduch: rucni rizeni" %
%   N7:64/2  PVZ_R %
%   N7:48/11  VYFUK  "Vyfuko- vani: rucni rizeni" %
%   N7:64/0  VY_R %
%   N7:48/12  ST_VYFUK  "Stabiliz. vyfukov.: rucni rizeni" %
%   N7:8/12  _STABILIZ  "Potvrzena predvolba" %
%   N7:64/1  SVY_R %
%   N7:48/13  ZACH_ZTRH  "Zachyt ztracene hlavy: rucni rizeni" %
%   N7:8/9  _HLAVA  "Potvrzena predvolba" %
%   N7:63/15  HZ_R %
%   N7:74/1  MOT_ZTRH  "Motor ztracene hlavy: rucni rizeni" %
%   N7:64/8  MH_R %
% Rung: 61 %
SOR XIC N7:74/0 BST XIC I:1.1/12 OTL N7:64/9 NXB XIC I:1.1/13 OTU N7:64/9 BND EOR
%   N7:74/0  ODJ_MASKY  "Odjisteni masky: rucni rizeni" %
%   I:1.1/12  NA_OT_VZ  "Nahoru, od sebe, vzad" %
%   N7:64/9  MODJ_R %
%   I:1.1/13  DO_ZA_VP  "Dolu, k sobe, vpred" %
% Rung: 62 %
SOR XIC N7:74/2 XIC N7:51/2 OTE N7:64/10 EOR
%   N7:74/2  NAPO_CO2  "CO2: rucni rizeni" %
%   N7:51/2  TLACITKA %
%   N7:64/10  CO2_R %

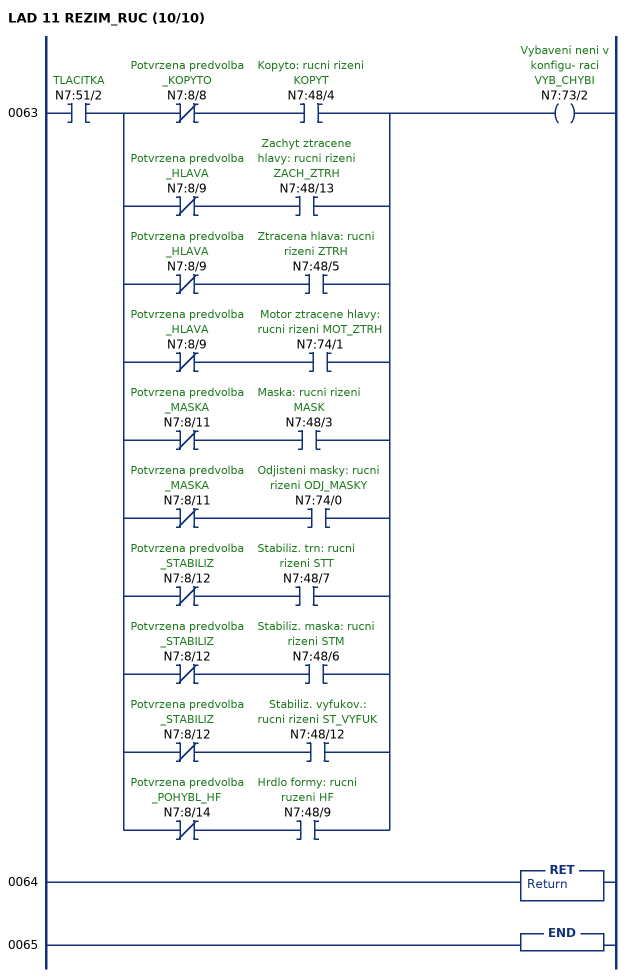
% Rung: 63 %
SOR XIC N7:51/2 BST XIO N7:8/8 XIC N7:48/4 NXB XIO N7:8/9 XIC N7:48/13 NXB XIO N7:8/9 XIC N7:48/5 NXB XIO N7:8/9 XIC N7:74/1 NXB XIO N7:8/11 XIC N7:48/3 NXB XIO N7:8/11 XIC N7:74/0 NXB XIO N7:8/12 XIC N7:48/7 NXB XIO N7:8/12 XIC N7:48/6 NXB XIO N7:8/12 XIC N7:48/12 NXB XIO N7:8/14 XIC N7:48/9 BND OTE N7:73/2 EOR
%   N7:51/2  TLACITKA %
%   N7:8/8  _KOPYTO  "Potvrzena predvolba" %
%   N7:48/4  KOPYT  "Kopyto: rucni rizeni" %
%   N7:8/9  _HLAVA  "Potvrzena predvolba" %
%   N7:48/13  ZACH_ZTRH  "Zachyt ztracene hlavy: rucni rizeni" %
%   N7:48/5  ZTRH  "Ztracena hlava: rucni rizeni" %
%   N7:74/1  MOT_ZTRH  "Motor ztracene hlavy: rucni rizeni" %
%   N7:8/11  _MASKA  "Potvrzena predvolba" %
%   N7:48/3  MASK  "Maska: rucni rizeni" %
%   N7:74/0  ODJ_MASKY  "Odjisteni masky: rucni rizeni" %
%   N7:8/12  _STABILIZ  "Potvrzena predvolba" %
%   N7:48/7  STT  "Stabiliz. trn: rucni rizeni" %
%   N7:48/6  STM  "Stabiliz. maska: rucni rizeni" %
%   N7:48/12  ST_VYFUK  "Stabiliz. vyfukov.: rucni rizeni" %
%   N7:8/14  _POHYBL_HF  "Potvrzena predvolba" %
%   N7:48/9  HF  "Hrdlo formy: rucni ruzeni" %
%   N7:73/2  VYB_CHYBI  "Vybaveni neni v konfigu- raci" %
% Rung: 64 %
SOR RET EOR
% Rung: 65 %
SOR END EOR

LADDER 12 "REZIM_VP"
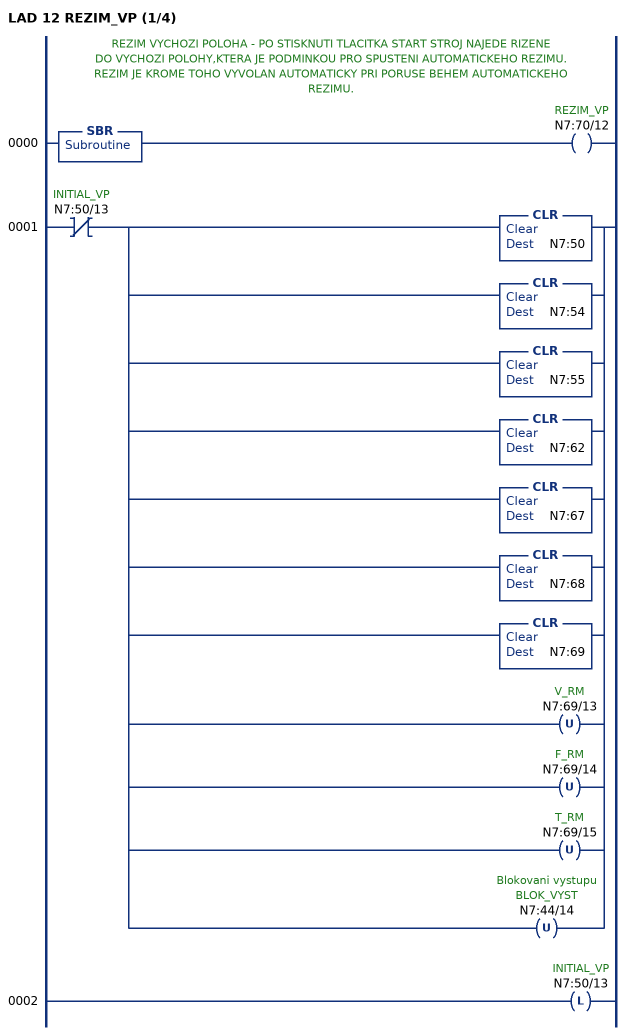
% Rung: 0 %
% REZIM VYCHOZI POLOHA - PO STISKNUTI TLACITKA START STROJ NAJEDE RIZENE
% DO VYCHOZI POLOHY,KTERA JE PODMINKOU PRO SPUSTENI AUTOMATICKEHO REZIMU.
% REZIM JE KROME TOHO VYVOLAN AUTOMATICKY PRI PORUSE BEHEM AUTOMATICKEHO
% REZIMU. %
SOR SBR OTE N7:70/12 EOR
%   N7:70/12  REZIM_VP %
% Rung: 1 %
SOR XIO N7:50/13 BST CLR N7:50 NXB CLR N7:54 NXB CLR N7:55 NXB CLR N7:62 NXB CLR N7:67 NXB CLR N7:68 NXB CLR N7:69 NXB OTU N7:69/13 NXB OTU N7:69/14 NXB OTU N7:69/15 NXB OTU N7:44/14 BND EOR
%   N7:50/13  INITIAL_VP %
%   CLR N7:50  "Pomocne merkry" %
%   CLR N7:54  "Logicke operandy casovacu" %
%   CLR N7:55  "Logicke operandy casovacu" %
%   CLR N7:62  "Merkry vystupu vychozi polohy" %
%   CLR N7:67  "Merkry vystupu automatic. rezimu" %
%   CLR N7:68  "Merkry vystupu automatic. rezimu" %
%   CLR N7:69  "Merkry vystupu automatic. rezimu, rampy" %
%   N7:69/13  V_RM %
%   N7:69/14  F_RM %
%   N7:69/15  T_RM %
%   N7:44/14  BLOK_VYST  "Blokovani vystupu" %
% Rung: 2 %
SOR OTL N7:50/13 EOR
%   N7:50/13  INITIAL_VP %

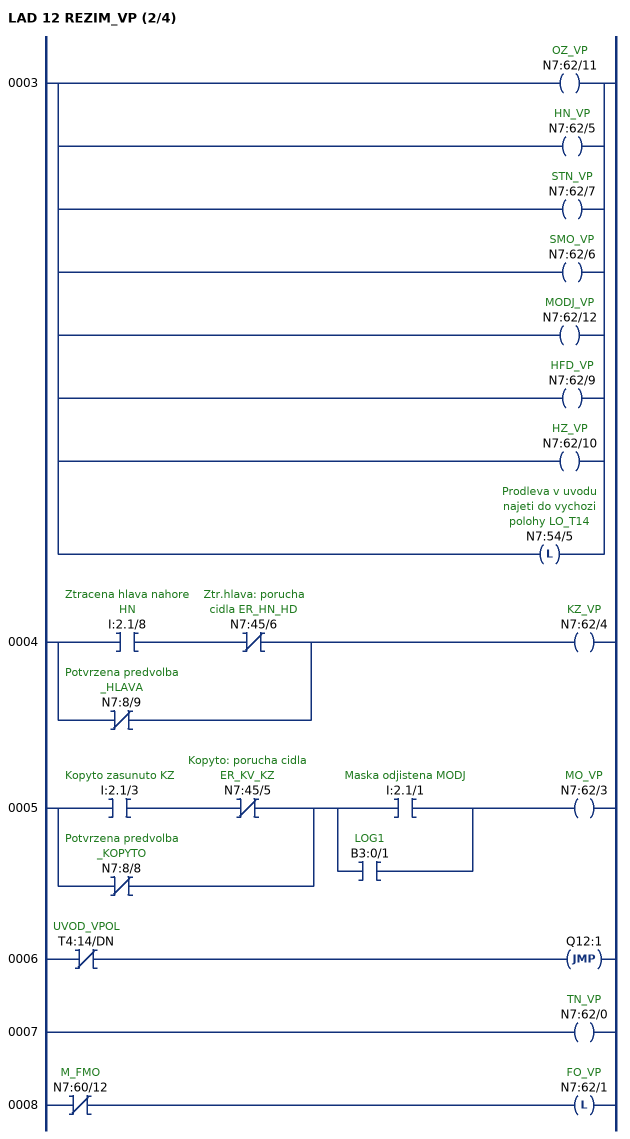
% Rung: 3 %
SOR BST OTE N7:62/11 NXB OTE N7:62/5 NXB OTE N7:62/7 NXB OTE N7:62/6 NXB OTE N7:62/12 NXB OTE N7:62/9 NXB OTE N7:62/10 NXB OTL N7:54/5 BND EOR
%   N7:62/11  OZ_VP %
%   N7:62/5  HN_VP %
%   N7:62/7  STN_VP %
%   N7:62/6  SMO_VP %
%   N7:62/12  MODJ_VP %
%   N7:62/9  HFD_VP %
%   N7:62/10  HZ_VP %
%   N7:54/5  LO_T14  "Prodleva v uvodu najeti do vychozi polohy" %
% Rung: 4 %
SOR BST XIC I:2.1/8 XIO N7:45/6 NXB XIO N7:8/9 BND OTE N7:62/4 EOR
%   I:2.1/8  HN  "Ztracena hlava nahore" %
%   N7:45/6  ER_HN_HD  "Ztr.hlava: porucha cidla" %
%   N7:8/9  _HLAVA  "Potvrzena predvolba" %
%   N7:62/4  KZ_VP %
% Rung: 5 %
SOR BST XIC I:2.1/3 XIO N7:45/5 NXB XIO N7:8/8 BND BST XIC I:2.1/1 NXB XIC B3:0/1 BND OTE N7:62/3 EOR
%   I:2.1/3  KZ  "Kopyto zasunuto" %
%   N7:45/5  ER_KV_KZ  "Kopyto: porucha cidla" %
%   N7:8/8  _KOPYTO  "Potvrzena predvolba" %
%   I:2.1/1  MODJ  "Maska odjistena" %
%   B3:0/1  LOG1 %
%   N7:62/3  MO_VP %
% Rung: 6 %
SOR XIO T4:14/DN JMP Q12:1 EOR
%   T4:14/DN  UVOD_VPOL %
% Rung: 7 %
SOR OTE N7:62/0 EOR
%   N7:62/0  TN_VP %
% Rung: 8 %
SOR XIO N7:60/12 OTL N7:62/1 EOR
%   N7:60/12  M_FMO %
%   N7:62/1  FO_VP %

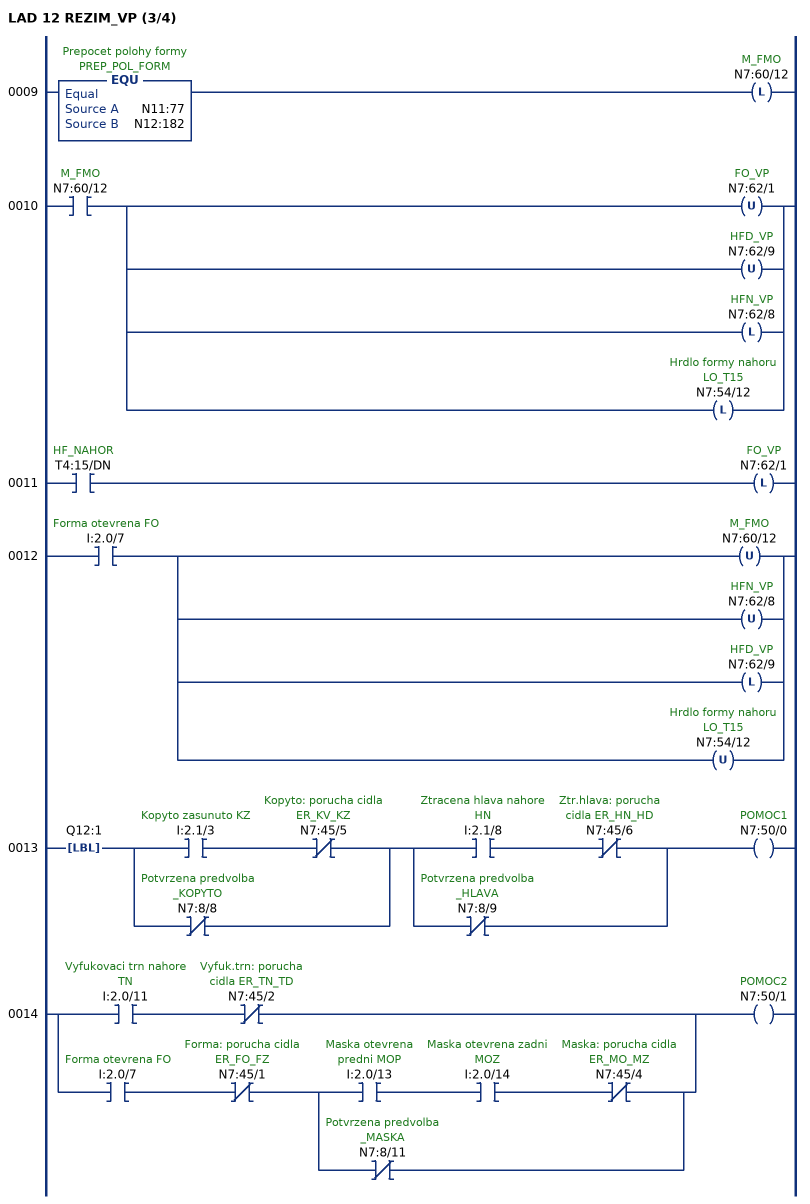
% Rung: 9 %
SOR EQU N11:77 N12:182 OTL N7:60/12 EOR
%   N11:77  PREP_POL_FORM  "Prepocet polohy formy" %
%   N7:60/12  M_FMO %
% Rung: 10 %
SOR XIC N7:60/12 BST OTU N7:62/1 NXB BST OTU N7:62/9 NXB OTL N7:62/8 NXB OTL N7:54/12 BND BND EOR
%   N7:60/12  M_FMO %
%   N7:62/1  FO_VP %
%   N7:62/9  HFD_VP %
%   N7:62/8  HFN_VP %
%   N7:54/12  LO_T15  "Hrdlo formy nahoru" %
% Rung: 11 %
SOR XIC T4:15/DN OTL N7:62/1 EOR
%   T4:15/DN  HF_NAHOR %
%   N7:62/1  FO_VP %
% Rung: 12 %
SOR XIC I:2.0/7 BST OTU N7:60/12 NXB OTU N7:62/8 NXB OTL N7:62/9 NXB OTU N7:54/12 BND EOR
%   I:2.0/7  FO  "Forma otevrena" %
%   N7:60/12  M_FMO %
%   N7:62/8  HFN_VP %
%   N7:62/9  HFD_VP %
%   N7:54/12  LO_T15  "Hrdlo formy nahoru" %
% Rung: 13 %
SOR LBL Q12:1 BST XIC I:2.1/3 XIO N7:45/5 NXB XIO N7:8/8 BND BST XIC I:2.1/8 XIO N7:45/6 NXB XIO N7:8/9 BND OTE N7:50/0 EOR
%   I:2.1/3  KZ  "Kopyto zasunuto" %
%   N7:45/5  ER_KV_KZ  "Kopyto: porucha cidla" %
%   N7:8/8  _KOPYTO  "Potvrzena predvolba" %
%   I:2.1/8  HN  "Ztracena hlava nahore" %
%   N7:45/6  ER_HN_HD  "Ztr.hlava: porucha cidla" %
%   N7:8/9  _HLAVA  "Potvrzena predvolba" %
%   N7:50/0  POMOC1 %
% Rung: 14 %
SOR BST XIC I:2.0/11 XIO N7:45/2 NXB XIC I:2.0/7 XIO N7:45/1 BST XIC I:2.0/13 XIC I:2.0/14 XIO N7:45/4 NXB XIO N7:8/11 BND BND OTE N7:50/1 EOR
%   I:2.0/11  TN  "Vyfukovaci trn nahore" %
%   N7:45/2  ER_TN_TD  "Vyfuk.trn: porucha cidla" %
%   I:2.0/7  FO  "Forma otevrena" %
%   N7:45/1  ER_FO_FZ  "Forma: porucha cidla" %
%   I:2.0/13  MOP  "Maska otevrena predni" %
%   I:2.0/14  MOZ  "Maska otevrena zadni" %
%   N7:45/4  ER_MO_MZ  "Maska: porucha cidla" %
%   N7:8/11  _MASKA  "Potvrzena predvolba" %
%   N7:50/1  POMOC2 %

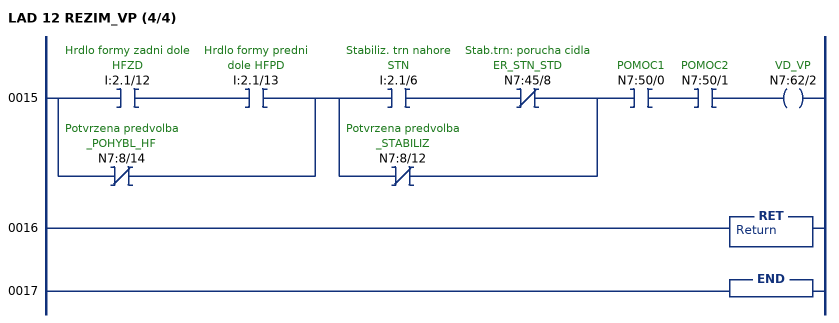
% Rung: 15 %
SOR BST XIC I:2.1/12 XIC I:2.1/13 NXB XIO N7:8/14 BND BST XIC I:2.1/6 XIO N7:45/8 NXB XIO N7:8/12 BND XIC N7:50/0 XIC N7:50/1 OTE N7:62/2 EOR
%   I:2.1/12  HFZD  "Hrdlo formy zadni dole" %
%   I:2.1/13  HFPD  "Hrdlo formy predni dole" %
%   N7:8/14  _POHYBL_HF  "Potvrzena predvolba" %
%   I:2.1/6  STN  "Stabiliz. trn nahore" %
%   N7:45/8  ER_STN_STD  "Stab.trn: porucha cidla" %
%   N7:8/12  _STABILIZ  "Potvrzena predvolba" %
%   N7:50/0  POMOC1 %
%   N7:50/1  POMOC2 %
%   N7:62/2  VD_VP %
% Rung: 16 %
SOR RET EOR
% Rung: 17 %
SOR END EOR

LADDER 13 "REZIM_AUT"
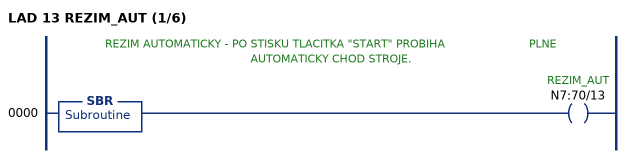
% Rung: 0 %
% REZIM AUTOMATICKY - PO STISKU TLACITKA "START" PROBIHA                        PLNE AUTOMATICKY CHOD STROJE. %
SOR SBR OTE N7:70/13 EOR
%   N7:70/13  REZIM_AUT %

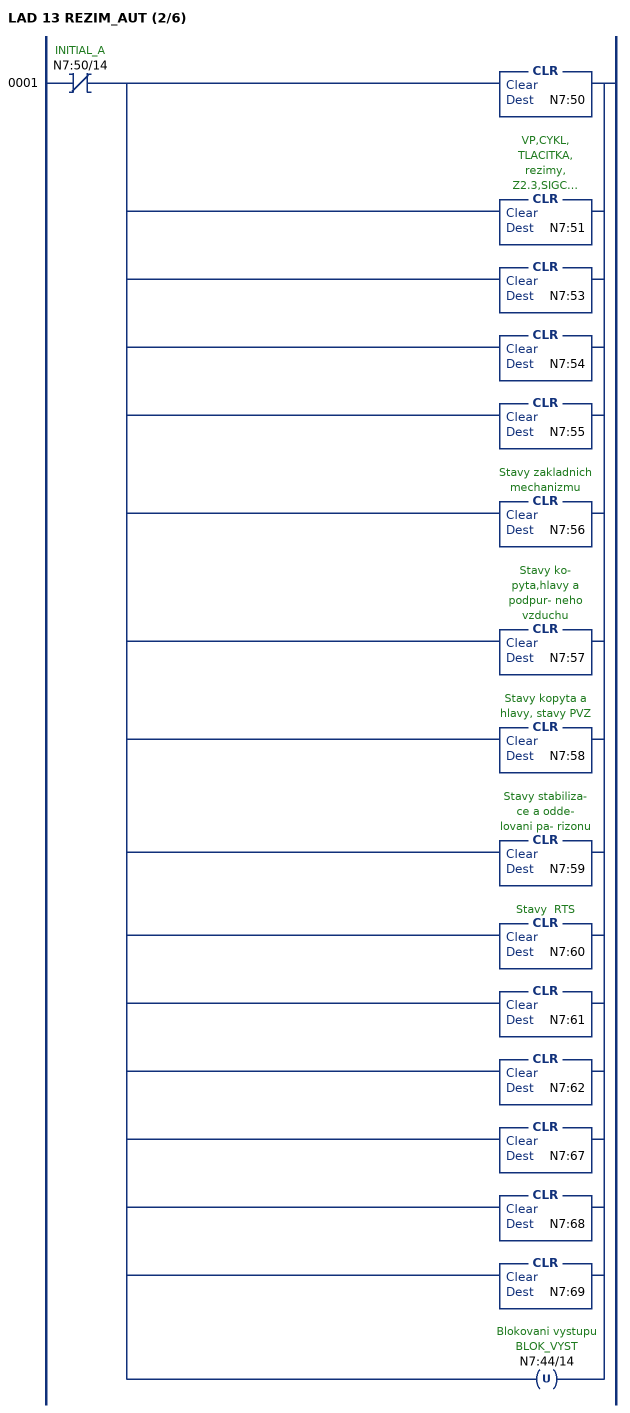
% Rung: 1 %
SOR XIO N7:50/14 BST CLR N7:50 NXB CLR N7:51 NXB CLR N7:53 NXB CLR N7:54 NXB CLR N7:55 NXB CLR N7:56 NXB CLR N7:57 NXB CLR N7:58 NXB CLR N7:59 NXB CLR N7:60 NXB CLR N7:61 NXB CLR N7:62 NXB CLR N7:67 NXB CLR N7:68 NXB CLR N7:69 NXB OTU N7:44/14 BND EOR
%   N7:50/14  INITIAL_A %
%   CLR N7:50  "Pomocne merkry" %
%   N7:51  "VP,CYKL, TLACITKA, rezimy, Z2.3,SIGCY DIAG,STAC" %
%   CLR N7:53  "Pameti automatic. rezimu" %
%   CLR N7:54  "Logicke operandy casovacu" %
%   CLR N7:55  "Logicke operandy casovacu" %
%   N7:56  "Stavy zakladnich mechanizmu" %
%   N7:57  "Stavy ko- pyta,hlavy a podpur- neho vzduchu" %
%   N7:58  "Stavy kopyta a hlavy, stavy PVZ" %
%   N7:59  "Stavy stabiliza- ce a odde- lovani pa- rizonu" %
%   N7:60  "Stavy  RTS" %
%   CLR N7:61  "Pameti automatic. rezimu" %
%   CLR N7:62  "Merkry vystupu vychozi polohy" %
%   CLR N7:67  "Merkry vystupu automatic. rezimu" %
%   CLR N7:68  "Merkry vystupu automatic. rezimu" %
%   CLR N7:69  "Merkry vystupu automatic. rezimu, rampy" %
%   N7:44/14  BLOK_VYST  "Blokovani vystupu" %

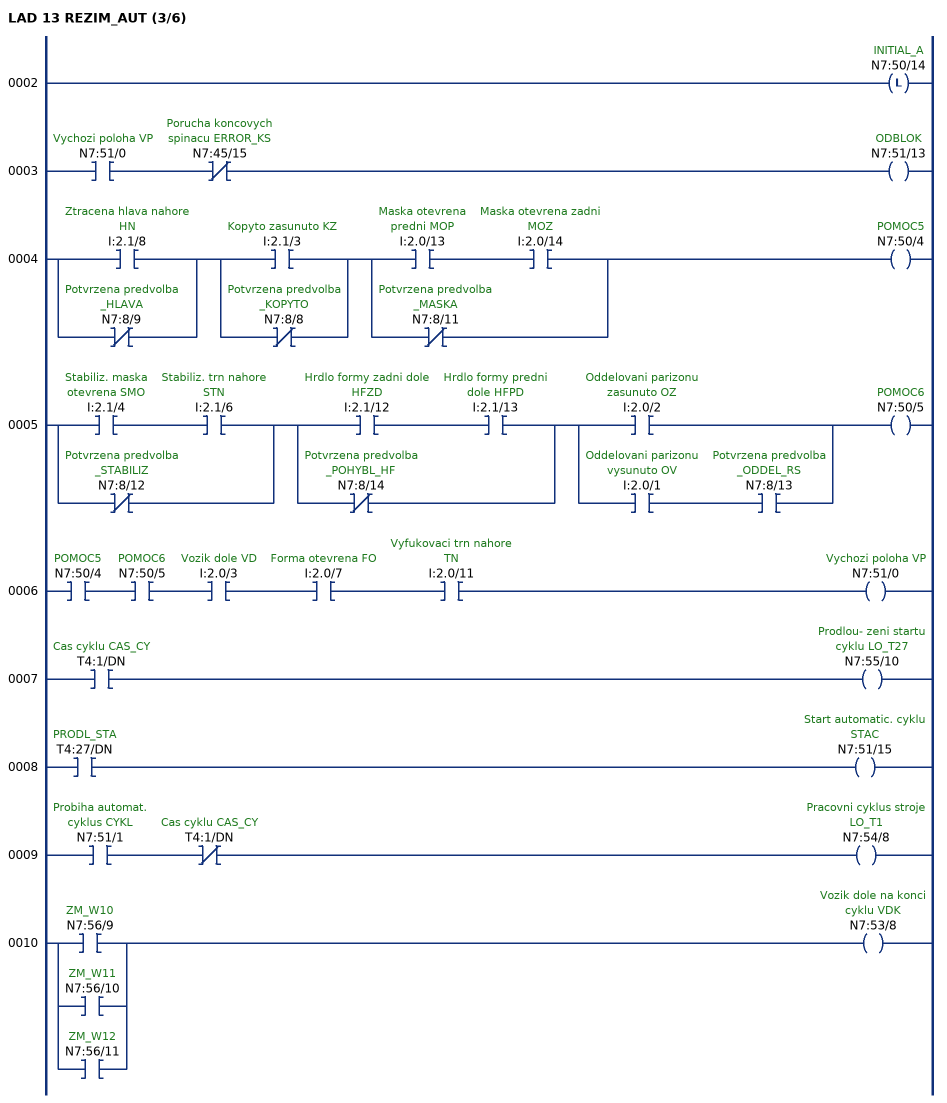
% Rung: 2 %
SOR OTL N7:50/14 EOR
%   N7:50/14  INITIAL_A %
% Rung: 3 %
SOR XIC N7:51/0 XIO N7:45/15 OTE N7:51/13 EOR
%   N7:51/0  VP  "Vychozi poloha" %
%   N7:45/15  ERROR_KS  "Porucha koncovych spinacu" %
%   N7:51/13  ODBLOK %
% Rung: 4 %
SOR BST XIC I:2.1/8 NXB XIO N7:8/9 BND BST XIC I:2.1/3 NXB XIO N7:8/8 BND BST XIC I:2.0/13 XIC I:2.0/14 NXB XIO N7:8/11 BND OTE N7:50/4 EOR
%   I:2.1/8  HN  "Ztracena hlava nahore" %
%   N7:8/9  _HLAVA  "Potvrzena predvolba" %
%   I:2.1/3  KZ  "Kopyto zasunuto" %
%   N7:8/8  _KOPYTO  "Potvrzena predvolba" %
%   I:2.0/13  MOP  "Maska otevrena predni" %
%   I:2.0/14  MOZ  "Maska otevrena zadni" %
%   N7:8/11  _MASKA  "Potvrzena predvolba" %
%   N7:50/4  POMOC5 %
% Rung: 5 %
SOR BST XIC I:2.1/4 XIC I:2.1/6 NXB XIO N7:8/12 BND BST XIC I:2.1/12 XIC I:2.1/13 NXB XIO N7:8/14 BND BST XIC I:2.0/2 NXB XIC I:2.0/1 XIC N7:8/13 BND OTE N7:50/5 EOR
%   I:2.1/4  SMO  "Stabiliz. maska otevrena" %
%   I:2.1/6  STN  "Stabiliz. trn nahore" %
%   N7:8/12  _STABILIZ  "Potvrzena predvolba" %
%   I:2.1/12  HFZD  "Hrdlo formy zadni dole" %
%   I:2.1/13  HFPD  "Hrdlo formy predni dole" %
%   N7:8/14  _POHYBL_HF  "Potvrzena predvolba" %
%   I:2.0/2  OZ  "Oddelovani parizonu zasunuto" %
%   I:2.0/1  OV  "Oddelovani parizonu vysunuto" %
%   N7:8/13  _ODDEL_RS  "Potvrzena predvolba" %
%   N7:50/5  POMOC6 %
% Rung: 6 %
SOR XIC N7:50/4 XIC N7:50/5 XIC I:2.0/3 XIC I:2.0/7 XIC I:2.0/11 OTE N7:51/0 EOR
%   N7:50/4  POMOC5 %
%   N7:50/5  POMOC6 %
%   I:2.0/3  VD  "Vozik dole" %
%   I:2.0/7  FO  "Forma otevrena" %
%   I:2.0/11  TN  "Vyfukovaci trn nahore" %
%   N7:51/0  VP  "Vychozi poloha" %
% Rung: 7 %
SOR XIC T4:1/DN OTE N7:55/10 EOR
%   T4:1/DN  CAS_CY  "Cas cyklu" %
%   N7:55/10  LO_T27  "Prodlou- zeni startu cyklu" %
% Rung: 8 %
SOR XIC T4:27/DN OTE N7:51/15 EOR
%   T4:27/DN  PRODL_STA %
%   N7:51/15  STAC  "Start automatic. cyklu" %
% Rung: 9 %
SOR XIC N7:51/1 XIO T4:1/DN OTE N7:54/8 EOR
%   N7:51/1  CYKL  "Probiha automat. cyklus" %
%   T4:1/DN  CAS_CY  "Cas cyklu" %
%   N7:54/8  LO_T1  "Pracovni cyklus stroje" %
% Rung: 10 %
SOR BST XIC N7:56/9 NXB XIC N7:56/10 NXB XIC N7:56/11 BND OTE N7:53/8 EOR
%   N7:56/9  ZM_W10 %
%   N7:56/10  ZM_W11 %
%   N7:56/11  ZM_W12 %
%   N7:53/8  VDK  "Vozik dole na konci cyklu" %

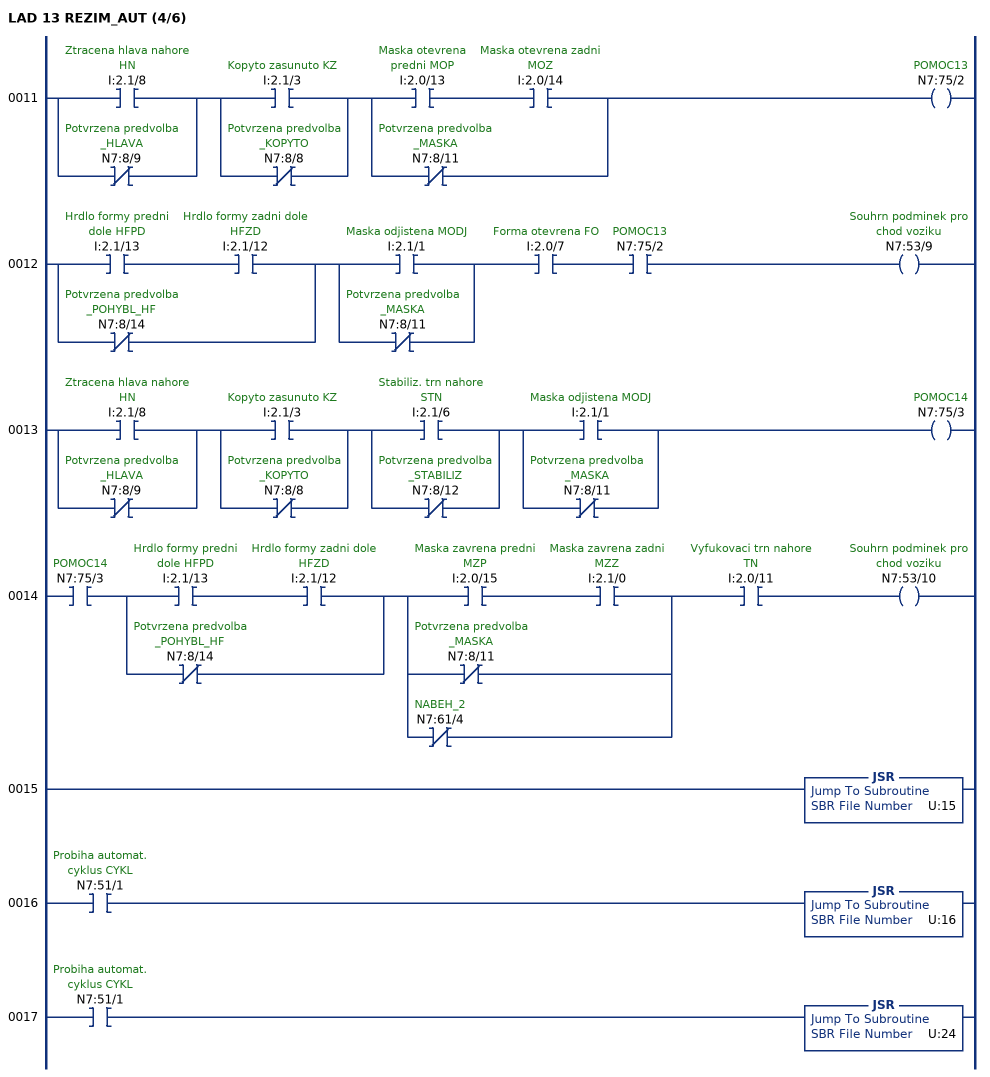
% Rung: 11 %
SOR BST XIC I:2.1/8 NXB XIO N7:8/9 BND BST XIC I:2.1/3 NXB XIO N7:8/8 BND BST XIC I:2.0/13 XIC I:2.0/14 NXB XIO N7:8/11 BND OTE N7:75/2 EOR
%   I:2.1/8  HN  "Ztracena hlava nahore" %
%   N7:8/9  _HLAVA  "Potvrzena predvolba" %
%   I:2.1/3  KZ  "Kopyto zasunuto" %
%   N7:8/8  _KOPYTO  "Potvrzena predvolba" %
%   I:2.0/13  MOP  "Maska otevrena predni" %
%   I:2.0/14  MOZ  "Maska otevrena zadni" %
%   N7:8/11  _MASKA  "Potvrzena predvolba" %
%   N7:75/2  POMOC13 %
% Rung: 12 %
SOR BST XIC I:2.1/13 XIC I:2.1/12 NXB XIO N7:8/14 BND BST XIC I:2.1/1 NXB XIO N7:8/11 BND XIC I:2.0/7 XIC N7:75/2 OTE N7:53/9 EOR
%   I:2.1/13  HFPD  "Hrdlo formy predni dole" %
%   I:2.1/12  HFZD  "Hrdlo formy zadni dole" %
%   N7:8/14  _POHYBL_HF  "Potvrzena predvolba" %
%   I:2.1/1  MODJ  "Maska odjistena" %
%   N7:8/11  _MASKA  "Potvrzena predvolba" %
%   I:2.0/7  FO  "Forma otevrena" %
%   N7:75/2  POMOC13 %
%   N7:53/9  "Souhrn podminek pro chod voziku" %
% Rung: 13 %
SOR BST XIC I:2.1/8 NXB XIO N7:8/9 BND BST XIC I:2.1/3 NXB XIO N7:8/8 BND BST XIC I:2.1/6 NXB XIO N7:8/12 BND BST XIC I:2.1/1 NXB XIO N7:8/11 BND OTE N7:75/3 EOR
%   I:2.1/8  HN  "Ztracena hlava nahore" %
%   N7:8/9  _HLAVA  "Potvrzena predvolba" %
%   I:2.1/3  KZ  "Kopyto zasunuto" %
%   N7:8/8  _KOPYTO  "Potvrzena predvolba" %
%   I:2.1/6  STN  "Stabiliz. trn nahore" %
%   N7:8/12  _STABILIZ  "Potvrzena predvolba" %
%   I:2.1/1  MODJ  "Maska odjistena" %
%   N7:8/11  _MASKA  "Potvrzena predvolba" %
%   N7:75/3  POMOC14 %
% Rung: 14 %
SOR XIC N7:75/3 BST XIC I:2.1/13 XIC I:2.1/12 NXB XIO N7:8/14 BND BST XIC I:2.0/15 XIC I:2.1/0 NXB XIO N7:8/11 NXB XIO N7:61/4 BND XIC I:2.0/11 OTE N7:53/10 EOR
%   N7:75/3  POMOC14 %
%   I:2.1/13  HFPD  "Hrdlo formy predni dole" %
%   I:2.1/12  HFZD  "Hrdlo formy zadni dole" %
%   N7:8/14  _POHYBL_HF  "Potvrzena predvolba" %
%   I:2.0/15  MZP  "Maska zavrena predni" %
%   I:2.1/0  MZZ  "Maska zavrena zadni" %
%   N7:8/11  _MASKA  "Potvrzena predvolba" %
%   N7:61/4  NABEH_2 %
%   I:2.0/11  TN  "Vyfukovaci trn nahore" %
%   N7:53/10  "Souhrn podminek pro chod voziku" %
% Rung: 15 %
SOR JSR U:15 EOR
%   JSR U:15  "START-STOP" %
% Rung: 16 %
SOR XIC N7:51/1 JSR U:16 EOR
%   N7:51/1  CYKL  "Probiha automat. cyklus" %
%   JSR U:16  "Zakladni mechanizmy" %
% Rung: 17 %
SOR XIC N7:51/1 JSR U:24 EOR
%   N7:51/1  CYKL  "Probiha automat. cyklus" %
%   JSR U:24  "Vyfukovaci trn" %

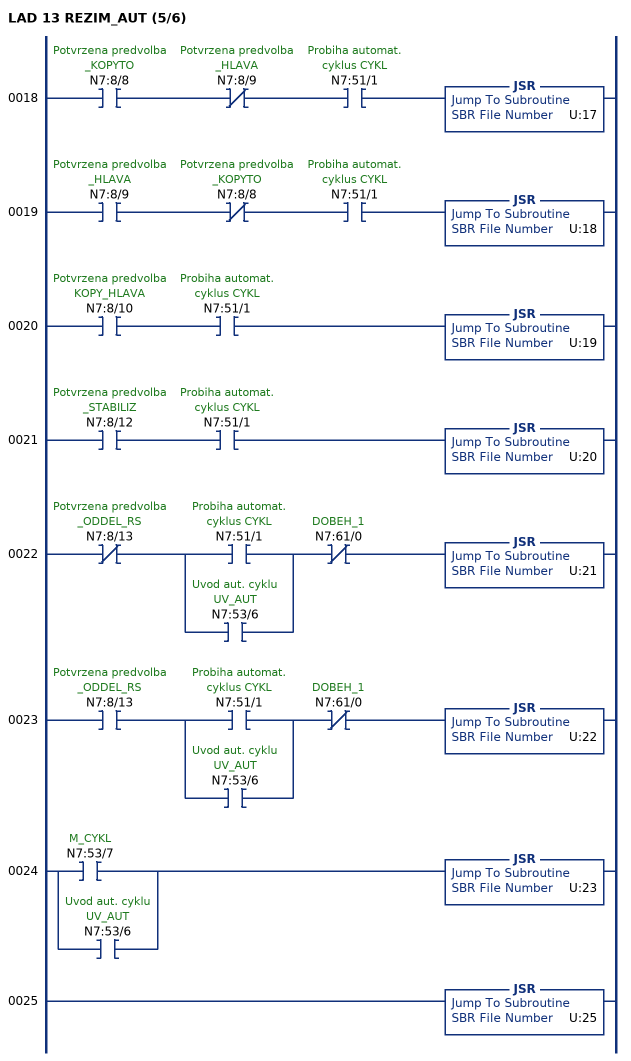
% Rung: 18 %
SOR XIC N7:8/8 XIO N7:8/9 XIC N7:51/1 JSR U:17 EOR
%   N7:8/8  _KOPYTO  "Potvrzena predvolba" %
%   N7:8/9  _HLAVA  "Potvrzena predvolba" %
%   N7:51/1  CYKL  "Probiha automat. cyklus" %
%   JSR U:17  "Kopyto solo" %
% Rung: 19 %
SOR XIC N7:8/9 XIO N7:8/8 XIC N7:51/1 JSR U:18 EOR
%   N7:8/9  _HLAVA  "Potvrzena predvolba" %
%   N7:8/8  _KOPYTO  "Potvrzena predvolba" %
%   N7:51/1  CYKL  "Probiha automat. cyklus" %
%   JSR U:18  "Hlava solo" %
% Rung: 20 %
SOR XIC N7:8/10 XIC N7:51/1 JSR U:19 EOR
%   N7:8/10  KOPY_HLAVA  "Potvrzena predvolba" %
%   N7:51/1  CYKL  "Probiha automat. cyklus" %
%   JSR U:19  "Kopyto a ztracena hlava" %
% Rung: 21 %
SOR XIC N7:8/12 XIC N7:51/1 JSR U:20 EOR
%   N7:8/12  _STABILIZ  "Potvrzena predvolba" %
%   N7:51/1  CYKL  "Probiha automat. cyklus" %
%   JSR U:20  "Stabili- zacni dochlazo- vani" %
% Rung: 22 %
SOR XIO N7:8/13 BST XIC N7:51/1 NXB XIC N7:53/6 BND XIO N7:61/0 JSR U:21 EOR
%   N7:8/13  _ODDEL_RS  "Potvrzena predvolba" %
%   N7:51/1  CYKL  "Probiha automat. cyklus" %
%   N7:53/6  UV_AUT  "Uvod aut. cyklu" %
%   N7:61/0  DOBEH_1 %
%   JSR U:21  "Oddelovani parizonu impulzni" %
% Rung: 23 %
SOR XIC N7:8/13 BST XIC N7:51/1 NXB XIC N7:53/6 BND XIO N7:61/0 JSR U:22 EOR
%   N7:8/13  _ODDEL_RS  "Potvrzena predvolba" %
%   N7:51/1  CYKL  "Probiha automat. cyklus" %
%   N7:53/6  UV_AUT  "Uvod aut. cyklu" %
%   N7:61/0  DOBEH_1 %
%   JSR U:22  "Oddelovani parizonu "RS"" %
% Rung: 24 %
SOR BST XIC N7:53/7 NXB XIC N7:53/6 BND JSR U:23 EOR
%   N7:53/7  M_CYKL %
%   N7:53/6  UV_AUT  "Uvod aut. cyklu" %
%   JSR U:23  "Podpurny vzduch" %
% Rung: 25 %
SOR JSR U:25 EOR
%   JSR U:25  "Chlazeni nadob pomoc CO2" %

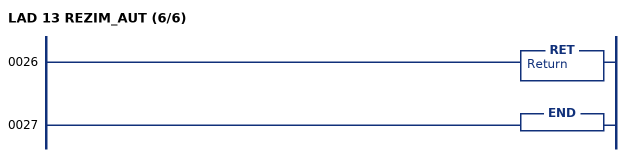
% Rung: 26 %
SOR RET EOR
% Rung: 27 %
SOR END EOR

LADDER 14 "REZIM_NULA"
